# B&R Automation Studio project NAEUL004C00R13L518F00 (part 48)

#### Act_Link.st - Change By Project
```iecst
(** 2019-07-04 **)
ACTION Act_Link:

	//Temporary (Recipe No Save)
	IF p_tyCurrProdRcp.sRcpNm = '' AND p_tyCurrProdRcp.diWidthInUM = 0 THEN
		p_tyCurrProdRcp	:= p_tyInternalReqProdRcp;
	END_IF

	//Info Message
	IF p_eLinkNtParamProjMag = ULMagDual THEN
		bBffrMagRemoved		:= (p_bLinkBffr1MagRemoved = TRUE) AND (p_bLinkBffr2MagRemoved = TRUE);
//		bOpsInitDone		:= ((p_bLinkNtParamProjMagConv1Prep AND p_bLinkOpsMagConvUL1InitDone) OR (NOT p_bLinkNtParamProjMagConv1Prep AND p_bLinkOpsMagUL1InitDone))
//								AND ((p_bLinkNtParamProjMagConv2Prep AND p_bLinkOpsMagConvUL2InitDone) OR (NOT p_bLinkNtParamProjMagConv2Prep AND p_bLinkOpsMagUL2InitDone));
		bOpsInitDone		:= p_bLinkOpsMagConvUL1InitDone AND p_bLinkOpsMagConvUL2InitDone;
	ELSIF p_eLinkNtParamProjMag = ULMagTriple THEN
		bBffrMagRemoved		:= (p_bLinkBffr1MagRemoved = TRUE) AND (p_bLinkBffr2MagRemoved = TRUE) AND (p_bLinkBffr3MagRemoved = TRUE);
//		bOpsInitDone		:= ((p_bLinkNtParamProjMagConv1Prep AND p_bLinkOpsMagConvUL1InitDone) OR (NOT p_bLinkNtParamProjMagConv1Prep AND p_bLinkOpsMagUL1InitDone))
//								AND ((p_bLinkNtParamProjMagConv2Prep AND p_bLinkOpsMagConvUL2InitDone) OR (NOT p_bLinkNtParamProjMagConv2Prep AND p_bLinkOpsMagUL2InitDone))
//								AND ((p_bLinkNtParamProjMagConv3Prep AND p_bLinkOpsMagConvUL3InitDone) OR (NOT p_bLinkNtParamProjMagConv3Prep AND p_bLinkOpsMagUL3InitDone));
		bOpsInitDone		:= p_bLinkOpsMagConvUL1InitDone AND p_bLinkOpsMagConvUL2InitDone AND p_bLinkOpsMagConvUL3InitDone;

	END_IF

	IF bBffrMagRemoved = FALSE THEN
		p_sInfoMsg		:= 'New Recipe Loaded';
		p_sInfoMsg		:= CONCAT(p_sInfoMsg , '$r$n');
		p_sInfoMsg		:= CONCAT(p_sInfoMsg , '$r$n');
		p_sInfoMsg		:= CONCAT(p_sInfoMsg , 'Please Remove All Magazines.');
	ELSE
		p_sInfoMsg		:= '';
	END_IF

	//Accept New Recipe Condition (Before Loaded New Recipe)
	p_bAccNewRcpCond	:=  bBffrMagRemoved = TRUE;

	//Update New Recipe Condition (After Loaded New Recipe)
	p_bUpdtNewRcpCond	:= TRUE;

	//Recipe Different
	p_bInternalReqProdRcpDiff	:= memcmp(ADR(p_tyCurrProdRcp) , ADR(p_tyInternalReqProdRcp) , SIZEOF(p_tyCurrProdRcp)) <> 0;
	p_bUpdtProdRcpDiff			:= memcmp(ADR(p_tyCurrProdRcp) , ADR(tyUpdtProdRcp) , SIZEOF(p_tyCurrProdRcp)) <> 0;

END_ACTION
```

#### Act_InitLocal.st - Do Not Change!!!
```iecst
(** 2020-08-06 **)
ACTION Act_InitLocal:

//Input Reference Link To Local Variable
	p_sMagRcpNm ACCESS ADR(sMagRcpNm);
	p_bUIProdAccData ACCESS ADR(bUIProdAccData);
	p_bUIProdUpdtData ACCESS ADR(bUIProdUpdtData);
	p_bUIMagAccData ACCESS ADR(bUIMagAccData);
	pa_tyProdRcpList ACCESS ADR(a_tyProdRcpList);
	p_tyCurrProdRcp ACCESS ADR(tyCurrProdRcp);
	p_sCurrMagRcpNm ACCESS ADR(sCurrMagRcpNm);
	p_bAccNewRcpCond ACCESS ADR(bAccNewRcpCond);
	p_bUpdtNewRcpCond ACCESS ADR(bUpdtNewRcpCond);
	p_bAutoUpdtData ACCESS ADR(bAutoUpdtData);
	p_sInfoMsg ACCESS ADR(sInfoMsg);
	p_bInternalUse ACCESS ADR(bInternalUse);
	p_tyInternalReqProdRcp ACCESS ADR(tyInternalReqProdRcp);
	p_bNewBrdEnteredCond ACCESS ADR(bNewBrdEnteredCond);
	p_bOldBrdExitedCond ACCESS ADR(bOldBrdExitedCond);
	p_bRlsBrd ACCESS ADR(bRlsBrd);
	p_bInternalReqProdRcpDiff ACCESS ADR(bInternalReqProdRcpDiff);
	p_bUpdtProdRcpDiff ACCESS ADR(bUpdtProdRcpDiff);
	p_bRlsBrdProdRcpDiff ACCESS ADR(bRlsBrdProdRcpDiff);
	p_tyFollower ACCESS ADR(tyFollower);

END_ACTION
```

#### Act_Background.st - Do Not Change!!!
```iecst
(** 2021-05-18 **)
ACTION Act_Background:

	IF p_bInternalUse = TRUE THEN
		tyLeaderToFollowerTag.sReqProdRcpNm		:= p_tyInternalReqProdRcp.sRcpNm;
		IF p_bWidth2Prep THEN
			tyLeaderToFollowerTag.diReqProdRcpWidth	:= p_tyInternalReqProdRcp.diWidthInUM2;
		ELSE
			tyLeaderToFollowerTag.diReqProdRcpWidth	:= p_tyInternalReqProdRcp.diWidthInUM;
		END_IF
		tyLeaderToFollowerTag.sReqMagRcpNm		:= '';
		tyLeaderToFollowerTag.bMnlAccData		:= FALSE;
		tyLeaderToFollowerTag.bBypassMnlAccData	:= FALSE;
		tyLeaderToFollowerTag.bBlkDS			:= FALSE;
		tyLeaderToFollowerTag.bBlkUS			:= FALSE;
		tyLeaderToFollowerTag.bBypassWidthChk	:= TRUE;
		tyLeaderToFollowerTag.bSetTm			:= FALSE;
		tyLeaderToFollowerTag.dtTm				:= 0;
		tyLeaderToFollowerTag.uiTmZone			:= 0;
		tyLeaderToFollowerTag.usiRunTm			:= 0;
		tyLeaderToFollowerTag.bProdNameUSWarn	:= FALSE;
		tyLeaderToFollowerTag.bProdNameDSWarn	:= FALSE;
		tyLeaderToFollowerTag.bProdWidthUSWarn	:= FALSE;
		tyLeaderToFollowerTag.bProdWidthDSWarn	:= FALSE;
		tyLeaderToFollowerTag.bLeaderSeqCtrlInActive	:= FALSE;
	END_IF

	Act_Background_UpdtData;

	//FB
	fbFollower.tyLeaderToFollowerTag	:= tyLeaderToFollowerTag;
	fbFollower.sMcNm					:= p_sMcNm;
	fbFollower.sIPAddr					:= p_sIPAddr;
	fbFollower.bSectionLeader			:= p_bSectionLeader;
	fbFollower.sCurrProdRcpNm			:= p_tyCurrProdRcp.sRcpNm;
	fbFollower.diCurrProdWidthUS		:= p_tyCurrProdRcp.diWidthInUM;
	fbFollower.diCurrProdWidthDS		:= p_tyCurrProdRcp.diWidthInUM2;
	fbFollower.sCurrMagRcpNm			:= p_sCurrMagRcpNm;
	fbFollower.sUpdtLeaderProdRcpNm		:= p_tyToLeaderProdRcp.sRcpNm;
	fbFollower.diUpdtLeaderProdWidthUS	:= p_tyToLeaderProdRcp.diWidthInUM;
	fbFollower.diUpdtLeaderProdWidthDS	:= p_tyToLeaderProdRcp.diWidthInUM2;
	fbFollower.sUpdtLeaderMagRcpNm		:= p_sMagRcpNm;
	fbFollower.bMnlAccDat				:= p_bMnlAccData;
	fbFollower.bAWEn					:= (p_bAWPrep = TRUE) AND (p_bAWDis = FALSE);
	fbFollower.bUSWidthChkEn			:= p_bUSWidthChkPrep AND p_bUSWidthChkEn;
	fbFollower.bUSWidthChkSen			:= p_bUSWidthChkSen;
	fbFollower.bDSWidthChkEn			:= p_bDSWidthChkPrep AND p_bDSWidthChkEn;
	fbFollower.bDSWidthChkSen			:= p_bDSWidthChkSen;
	fbFollower.bProdWidthChk			:= p_bProdWidthChk;
	fbFollower.bProdRcpErr				:= bProdRcpErr;
	fbFollower.bMagRcpErr				:= bMagRcpErr;
	fbFollower.bSetTmErr				:= bSetTmErr;
	fbFollower.eCurrMachineStat			:= eCurrMachineStat;
	fbFollower.bProdChgOverActive		:= (p_eAWStat = AWActGoWidthOff);
	fbFollower.bDBAOnWOAlign			:= p_bDBAOnWOAlign;
	fbFollower(bEn := TRUE);

	tyFollowerToLeaderTag	:= fbFollower.tyFollowerToLeaderTag;
	bProdAccDataReq			:= fbFollower.bProdAccDataReq OR (p_bInternalReqProdRcpDiff = TRUE) ;
	bMagAccDataReq			:= fbFollower.bMagAccDataReq;
	bAutoAccData			:= fbFollower.bAutoAccData;

	IF p_bInternalUse THEN
		bLeaderOnline		:= TRUE;
	ELSE
		bLeaderOnline		:= tyLeaderInfo.bOnline;
	END_IF

	IF bLeaderOnline=FALSE THEN
		bUSAllow				:= TRUE;
		bDSAllow				:= TRUE;
		bLeaderSeqCtrlInActive	:= FALSE;
	ELSE
		bUSAllow				:= fbFollower.bUSAllow AND (p_bInternalReqProdRcpDiff = FALSE);
		bDSAllow				:= fbFollower.bDSAllow;
		bLeaderSeqCtrlInActive	:= tyLeaderToFollowerTag.bLeaderSeqCtrlInActive;
	END_IF

	fbOnlineChk.tyLeaderToFollowerTag	:= tyLeaderToFollowerTag;
	fbOnlineChk(bEn := TRUE);

	Act_Background_AccData;
	Act_Background_ChkRlsBrd;

	//Set Time
	IF EDGEPOS(tyLeaderToFollowerTag.bSetTm) THEN
		bSetTm	:= TRUE;
	END_IF

	IF bSetTm = TRUE THEN
		eTimeAct	:= TimeActSetTime;

		IF (p_eTimeStat = TimeActSetTime) AND (p_eTimeStatus = Done) THEN
			eTimeAct		:= TimeActIdle;
			bSetTm			:= FALSE;
		ELSIF p_eTimeStatus = Error THEN
			eTimeAct		:= TimeActIdle;
			bSetTm			:= FALSE;
		END_IF
	END_IF

	bSetTmErr	:= p_eTimeStatus = Error;

	IF (eStatus = Error) AND bRstErr THEN
		eStatus		:= Idle;
		udiStatus	:= 0;
		bProdRcpErr	:= FALSE;
		bProdRcpErrNotExist	:= FALSE;
		bProdRcpErrWidthMismatch:= FALSE;
		bMagRcpErr	:= FALSE;
	END_IF

END_ACTION
```

#### Act_Background_ChkRlsBrd.st - Do Not Change!!!
```iecst
ACTION Act_Background_ChkRlsBrd:

	IF tyRlsBrdProdRcpNm.sRcpNm = '' THEN
		tyRlsBrdProdRcpNm	:= p_tyCurrProdRcp;

	ELSIF (tyRlsBrdProdRcpNm.sRcpNm <> p_tyCurrProdRcp.sRcpNm) OR (p_bRlsBrdProdRcpDiff = TRUE) THEN

		IF p_bNewBrdEnteredCond = TRUE THEN
			bNewBrdEntered	:= TRUE;
		END_IF

		IF p_bOldBrdExitedCond = TRUE THEN
			bOldBrdExited	:= TRUE;
		END_IF

		IF bNewBrdEntered AND bOldBrdExited THEN
			tylocalFollower.Out.bWaitRlsBrd	:= TRUE;
		END_IF

		IF tylocalFollower.Out.bWaitRlsBrd AND p_bRlsBrd THEN
			tyRlsBrdProdRcpNm	:= p_tyCurrProdRcp;
		END_IF

	ELSE
		bNewBrdEntered	:= FALSE;
		bOldBrdExited	:= FALSE;
		tylocalFollower.Out.bWaitRlsBrd		:= FALSE;

	END_IF

END_ACTION
```

#### Act_Background_AccData.st - Do Not Change!!!
```iecst
ACTION Act_Background_AccData:
	//Product Accept Data Request
	CASE usiProdAccDatStep OF
		0:
			//Check Error & Request Accept Data
			// If Product Name/Width Error, Check In Background To Update Data
			IF ((tylocalFollower.Out.eStatus <> Error) AND (bProdAccDataReq = TRUE)) OR bProdRcpErr THEN
				sReqProdRcpNm		:= tyLeaderToFollowerTag.sReqProdRcpNm;
				diReqProdRcpWidth	:= tyLeaderToFollowerTag.diReqProdRcpWidth;
				usiProdAccDatStep	:= 1;
			END_IF

			IF bLeaderOnline=FALSE THEN
				tyInfoData.udiCode		:= 0;
				tyInfoData.eSeverity	:= AlmSeverityNA;

				bProdRcpErr 			:= FALSE;
				bProdRcpErrNotExist		:= FALSE;
				bProdRcpErrWidthMismatch:= FALSE;
			END_IF

		1:
			IF p_bInternalUse THEN
				usiProdAccDatStep	:= 2;
			ELSE

				//Check In List Of Recipe
				FOR i := 1 TO 2000 DO
					IF sReqProdRcpNm = '' THEN
						EXIT;
					ELSIF sReqProdRcpNm = pa_tyProdRcpList[i].sRcpNm  THEN
						EXIT;
					END_IF
				END_FOR

				IF sReqProdRcpNm = pa_tyProdRcpList[i].sRcpNm AND diReqProdRcpWidth <> pa_tyProdRcpList[i].diWidthInUM THEN
					//Width Mismatch
					bProdRcpErr := TRUE;
					bProdRcpErrWidthMismatch:= TRUE;
					bProdRcpErrNotExist		:= FALSE;
					usiProdAccDatStep	:= 0;
				ELSIF i > 2000 THEN
					//Recipe Not Exist
					bProdRcpErr := TRUE;
					bProdRcpErrNotExist	:= TRUE;
					bProdRcpErrWidthMismatch:= FALSE;
					usiProdAccDatStep	:= 0;
				ELSE
					bProdRcpErr := FALSE;
					bProdRcpErrNotExist	:= FALSE;
					bProdRcpErrWidthMismatch:= FALSE;
					usiProdAccDatStep	:= 2;
				END_IF

				//Info Message
				IF bLeaderOnline=FALSE THEN
					tyInfoData.udiCode		:= 0;
					tyInfoData.eSeverity	:= AlmSeverityNA;

					bProdRcpErr 			:= FALSE;
					bProdRcpErrNotExist		:= FALSE;
					bProdRcpErrWidthMismatch:= FALSE;
				ELSE
					IF p_bInternalUse = FALSE THEN
						IF bLeaderInfo OR bFollowerInfo THEN
//							tyInfoData.sProgNm		:= g_tyNtParamCurr.sFollower1ProgNm;
							tyInfoData.udiCode		:= 10000;
							tyInfoData.eSeverity	:= AlmSeverityInfo;
						ELSE
//							tyInfoData.sProgNm		:= '';
							tyInfoData.udiCode		:= 0;
							tyInfoData.eSeverity	:= AlmSeverityNA;
						END_IF
					ELSE
						IF p_sInfoMsg <> '' THEN
//							tyInfoData.sProgNm		:= g_tyNtParamCurr.sFollower1ProgNm;
							tyInfoData.udiCode		:= 10000;
							tyInfoData.eSeverity	:= AlmSeverityInfo;
						ELSE
//							tyInfoData.sProgNm		:= '';
							tyInfoData.udiCode		:= 0;
							tyInfoData.eSeverity	:= AlmSeverityNA;
							tyInfoData.sAlmMsg		:= '';
						END_IF
					END_IF
				END_IF
			END_IF

		2:
			//Manual Accept Data Check
			IF bProdAccDataReq = TRUE THEN
				IF bAutoAccData = FALSE THEN
				tylocalFollower.Out.bProdAccDataMnl	:= TRUE;

					//Info Message
					IF bLeaderOnline=FALSE THEN
//						tyInfoData.sProgNm		:= '';
						tyInfoData.udiCode		:= 0;
						tyInfoData.eSeverity	:= AlmSeverityNA;
//						tyInfoData.sAlmMsg		:= '';
					ELSE
						IF p_sInfoMsg <> '' THEN
//							tyInfoData.sProgNm		:= g_tyNtParamCurr.sFollower1ProgNm;
							tyInfoData.udiCode		:= 10000;
							tyInfoData.eSeverity	:= AlmSeverityInfo;
//							tyInfoData.sAlmMsg		:= p_sInfoMsg;
						ELSE
//							tyInfoData.sProgNm		:= '';
							tyInfoData.udiCode		:= 0;
							tyInfoData.eSeverity	:= AlmSeverityNA;
//							tyInfoData.sAlmMsg		:= '';
						END_IF
					END_IF

					IF p_bUIProdAccData = TRUE THEN
						tylocalFollower.Out.bProdAccDataMnl		:= FALSE;
						usiProdAccDatStep	:= 3;
					END_IF
				ELSE
					bProdAccDataMnl		:= FALSE;
					tylocalFollower.Out.bProdAccDataMnl		:= FALSE;
					usiProdAccDatStep	:= 3;
				END_IF
			ELSE
				bProdAccDataMnl		:= FALSE;
				usiProdAccDatStep	:= 6;
			END_IF

		3:
			//Accept New Recipe Condition
			IF bProdAccDataReq = TRUE THEN
				IF p_bAccNewRcpCond = TRUE THEN

					usiProdAccDatStep	:= 4;
				ELSE
					//Info Message
					IF bLeaderOnline=FALSE THEN
//						tyInfoData.sProgNm		:= '';
						tyInfoData.udiCode		:= 0;
						tyInfoData.eSeverity	:= AlmSeverityNA;
//						tyInfoData.sAlmMsg		:= '';
					ELSE
						IF p_sInfoMsg <> '' THEN
//							tyInfoData.sProgNm		:= g_tyNtParamCurr.sFollower1ProgNm;
							tyInfoData.udiCode		:= 10000;
							tyInfoData.eSeverity	:= AlmSeverityInfo;
//							tyInfoData.sAlmMsg		:= p_sInfoMsg;
						ELSE
//							tyInfoData.sProgNm		:= '';
							tyInfoData.udiCode		:= 0;
							tyInfoData.eSeverity	:= AlmSeverityNA;
//							tyInfoData.sAlmMsg		:= '';
						END_IF
					END_IF
				END_IF
			ELSE
				usiProdAccDatStep	:= 6;
			END_IF

		4:
			//Accept New Recipe Name
			IF p_bInternalUse = TRUE THEN

				p_tyCurrProdRcp	:= p_tyInternalReqProdRcp;
				usiProdAccDatStep := 6;
			ELSE

				FOR i := 1 TO 2000 DO
					IF sReqProdRcpNm = '' THEN
						EXIT;
					ELSIF sReqProdRcpNm = pa_tyProdRcpList[i].sRcpNm THEN
						p_tyCurrProdRcp	:= pa_tyProdRcpList[i];
						EXIT;
					END_IF
				END_FOR

				IF i > 2000 THEN
					//Recipe Not Exist
					bProdRcpErr := TRUE;
					bProdRcpErrNotExist	:= TRUE;
				END_IF
				usiProdAccDatStep	:= 5;
			END_IF

		5:
			(* Add *)
			p_tyProdRcpCurrRcpWr 	:= p_tyCurrProdRcp;
			p_eLinkUIProdRcpAct 	:= ProdRcpActWriteCurrRcpParam;

			IF p_eProdRcpStat = ProdRcpActWriteCurrRcpParam AND p_eProdRcpStatus = Done THEN
				p_eLinkUIProdRcpAct := ProdRcpActIdle;
				usiProdAccDatStep := 6;
			END_IF

		6:
			//Clear Info Message
			tyInfoData.sProgNm		:= '';
			tyInfoData.udiCode		:= 0;
			tyInfoData.eSeverity	:= AlmSeverityNA;
			tyInfoData.sAlmMsg		:= '';

			usiProdAccDatStep	:= 0;

	END_CASE

END_ACTION
```

#### Act_Main_Disable.st - Do Not Change!!!
```iecst
ACTION Act_Main_Disable:

	tylocalFollower.Out.bUSAllow			:= TRUE;
	tylocalFollower.Out.bDSAllow			:= TRUE;
	tylocalFollower.Out.bProdAccDataMnl		:= FALSE;
	tylocalFollower.Out.bProdUpdtDataMnl	:= FALSE;
	tylocalFollower.Out.bMagAccDataMnl		:= FALSE;
	tylocalFollower.Out.bWaitRlsBrd			:= FALSE;

	usiProdAccDatStep		:= 0;
	usiProdUpdtDatStep		:= 0;
	tyInfoData.udiCode		:= 0;
	tyInfoData.eSeverity	:= AlmSeverityNA;

	usiMagAccDatStep		:= 0;
	tylocalFollower.Out.tyInfoData1.udiCode		:= 0;
	tylocalFollower.Out.tyInfoData1.eSeverity	:= AlmSeverityNA;

	bSetTm		:= FALSE;

	tylocalFollower.Out.eStatus		:= Idle;
	udiStatus	:= 0;
	bProdRcpErr	:= FALSE;
	bMagRcpErr	:= FALSE;
	tylocalFollower.Out.bLdrSeqCtrlInActive	:= FALSE;

	bProdRcpErrNotExist		:= FALSE;
	bProdRcpErrWidthMismatch:= FALSE;

END_ACTION
```

#### Act_Alarm.st - Do Not Change!!!
```iecst
ACTION Act_Alarm:

	IF g_tyRstErrOut.udiRstErr <> udiRstErrOld THEN
		bRstErr			:= TRUE;
		udiRstErrOld	:= g_tyRstErrOut.udiRstErr;
	ELSE
		bRstErr			:= FALSE;
	END_IF

	//Error
	IF EDGEPOS(tylocalFollower.Out.eStatus = Error) THEN

		tylocalFollower.Out.tyAlmData.udiCode		:= udiStatus;
		tylocalFollower.Out.tyAlmData.eSeverity		:= AlmSeverityError;
		tylocalFollower.Out.tyAlmData.udiRunTime	:= tyAlmData.udiRunTime + 1;
		tylocalFollower.Out.tyAlmData.bAlm			:= TRUE;
		tylocalFollower.Out.tyAlmData.udiModuleNum	:= udiModuleNum;
		g_tyAlmProgNm.sLFFollowerProgNm				 := g_tyNtParamCurr.sFollower2ProgNm;

	ELSIF bRstErr AND (tylocalFollower.Out.tyAlmData.udiCode <> 0) THEN

		tylocalFollower.Out.tyAlmData.udiCode	:= 0;
		tylocalFollower.Out.tyAlmData.eSeverity	:= AlmSeverityNA;
		tylocalFollower.Out.tyAlmData.bAlm		:= FALSE;

	END_IF

END_ACTION
```

#### InputRef.var - Do Not Change!!!
```iecst
(*2020-08-06*)
(**)
(*General*)
VAR
	p_udiRstErr : REFERENCE TO UDINT;
	p_bPrep : REFERENCE TO BOOL;
	p_bEn : REFERENCE TO BOOL;
	p_bDis : REFERENCE TO BOOL;
END_VAR
(**)
(*Configuration*)
VAR
	p_eAWStat : REFERENCE TO eAWAction;
	p_sIPAddr : REFERENCE TO STRING[15];
END_VAR
(**)
(*Input*)
VAR
	p_sMcNm : REFERENCE TO STRING[30];
	p_bAWPrep : REFERENCE TO BOOL;
	p_bAWDis : REFERENCE TO BOOL;
	p_bMnlAccData : REFERENCE TO BOOL;
	p_bSectionLeader : REFERENCE TO BOOL;
	p_sMagRcpNm : REFERENCE TO STRING[30];
	p_diWidthLimit : REFERENCE TO DINT;
	p_bWidth2Prep : REFERENCE TO BOOL;
	p_bNtParamAutoRcpPrep : REFERENCE TO BOOL;
	p_bMcParamAutoRcpDis : REFERENCE TO BOOL;
	p_bNtParamAutoRcpF1ArbitraryType : REFERENCE TO BOOL;
	p_bUSWidthChkPrep : REFERENCE TO BOOL;
	p_bUSWidthChkEn : REFERENCE TO BOOL;
	p_bUSWidthChkSen : REFERENCE TO BOOL;
	p_bDSWidthChkPrep : REFERENCE TO BOOL;
	p_bDSWidthChkEn : REFERENCE TO BOOL;
	p_bDSWidthChkSen : REFERENCE TO BOOL;
	p_bProdWidthChk : REFERENCE TO BOOL;
	p_bUIProdAccData : REFERENCE TO BOOL;
	p_bUIProdUpdtData : REFERENCE TO BOOL;
	p_bUIMagAccData : REFERENCE TO BOOL;
	pa_tyProdRcpList : REFERENCE TO ARRAY[1..c_udiProdRcpMax] OF tyProdRcpParam;
	p_tyCurrProdRcp : REFERENCE TO tyProdRcpParam;
	p_sCurrMagRcpNm : REFERENCE TO STRING[30];
	p_eTimeStat : REFERENCE TO eTimeAction;
	p_eTimeStatus : REFERENCE TO eFBStatus;
	p_bAccNewRcpCond : REFERENCE TO BOOL;
	p_bUpdtNewRcpCond : REFERENCE TO BOOL;
	p_bAutoUpdtData : REFERENCE TO BOOL;
	p_sInfoMsg : REFERENCE TO STRING[200];
	p_bInternalUse : REFERENCE TO BOOL;
	p_tyInternalReqProdRcp : REFERENCE TO tyProdRcpParam;
	p_bNewBrdEnteredCond : REFERENCE TO BOOL;
	p_bOldBrdExitedCond : REFERENCE TO BOOL;
	p_bRlsBrd : REFERENCE TO BOOL;
	p_tyToLeaderProdRcp : REFERENCE TO tyProdRcpParam;
	p_bInternalReqProdRcpDiff : REFERENCE TO BOOL;
	p_bUpdtProdRcpDiff : REFERENCE TO BOOL;
	p_bRlsBrdProdRcpDiff : REFERENCE TO BOOL;
	p_sProgNm : REFERENCE TO STRING[15];
	p_bNtSettingsLoadDone : REFERENCE TO BOOL;
	p_tOnlineChkDlyTm : REFERENCE TO TIME;
	p_bManual : REFERENCE TO BOOL;
	p_bErr : REFERENCE TO BOOL;
	p_bWarning : REFERENCE TO BOOL;
	p_bOps : REFERENCE TO BOOL;
	p_bStandby : REFERENCE TO BOOL;
	p_bDBAOnWOAlign : REFERENCE TO BOOL;
END_VAR
```

#### Local.var - Do Not Change!!!
```iecst
VAR
	tylocalFollower : tyLFFollower1;
END_VAR
(**)
VAR
	udiStatus : UDINT := 0;
END_VAR
(**)
(*Local Alarm*)
VAR
	tyAlmData : tyAlmDat;
	tyInfoData : tyAlmDat;
	tyInfoData1 : tyAlmDat;
END_VAR
(**)
VAR
	sMagRcpNm : STRING[30];
	bUIProdAccData : BOOL;
	bUIProdUpdtData : BOOL;
	bUIMagAccData : BOOL;
	a_tyProdRcpList : ARRAY[1..c_udiProdRcpMax] OF tyProdRcpParam;
	tyDispProdRcp : tyProdRcpParam;
	tyCurrProdRcp : tyProdRcpParam;
	sCurrMagRcpNm : STRING[30];
	bAccNewRcpCond : BOOL;
	bUpdtNewRcpCond : BOOL;
	bAutoUpdtData : BOOL;
	sInfoMsg : STRING[200];
	bInternalUse : BOOL;
	tyInternalReqProdRcp : tyProdRcpParam;
	bNewBrdEnteredCond : BOOL;
	bOldBrdExitedCond : BOOL;
	bRlsBrd : BOOL;
	tyToLeaderProdRcp : tyProdRcpParam;
	bInternalReqProdRcpDiff : BOOL;
	bUpdtProdRcpDiff : BOOL;
	bRlsBrdProdRcpDiff : BOOL;
	sWidthInUMTemp : STRING[80];
END_VAR
(**)
(*Local*)
VAR
	bRstErr : BOOL;
	udiRstErrOld : UDINT;
	bInitDone : BOOL;
	bInitialDone : BOOL;
	bAutoAccData : BOOL;
	bProdRcpErr : BOOL;
	bMagRcpErr : BOOL;
	bSetTmErr : BOOL;
	bProdAccDataReq : BOOL;
	sReqProdRcpNm : STRING[254];
	diReqProdRcpWidth : DINT;
	bMagAccDataReq : BOOL;
	sReqMagRcpNm : STRING[30];
	usiProdAccDatStep : USINT;
	usiMagAccDatStep : USINT;
	usiProdUpdtDatStep : USINT;
	tyRlsBrdProdRcpNm : tyProdRcpParam;
	bNewBrdEntered : BOOL;
	bOldBrdExited : BOOL;
	i : INT;
	bSetTm : BOOL;
	fbOnlineChk : fbLFFollowerOnlineChk;
	fbFollower : fbLFFollower;
	tyLeaderToFollowerTag : tyLFLeaderToFollowerTag;
	tyFollowerToLeaderTag : tyLFFollowerToLeaderTag;
	eCurrMachineStat : eMachineStat;
	bLeaderOnline : BOOL;
	bLeaderInfo : BOOL;
	bFollowerInfo : BOOL;
	bProdRcpErrNotExist : BOOL;
	bProdRcpErrWidthMismatch : BOOL;
	tyFollower : {REDUND_UNREPLICABLE} tyLFFollowerOut1;
	bBffrMagRemoved : BOOL;
	bOpsInitDone : BOOL;
END_VAR
(**)
VAR
	p_sMagRcpNm : REFERENCE TO STRING[30];
	p_bUIProdAccData : REFERENCE TO BOOL;
	p_bUIProdUpdtData : REFERENCE TO BOOL;
	p_bUIMagAccData : REFERENCE TO BOOL;
	pa_tyProdRcpList : REFERENCE TO ARRAY[1..c_udiProdRcpMax] OF tyProdRcpParam;
	p_tyCurrProdRcp : REFERENCE TO tyProdRcpParam;
	p_tyDispProdRcp : REFERENCE TO tyProdRcpParam;
	p_sCurrMagRcpNm : REFERENCE TO STRING[30];
	p_bAccNewRcpCond : REFERENCE TO BOOL;
	p_bUpdtNewRcpCond : REFERENCE TO BOOL;
	p_bAutoUpdtData : REFERENCE TO BOOL;
	p_sInfoMsg : REFERENCE TO STRING[200];
	p_bInternalUse : REFERENCE TO BOOL;
	p_tyInternalReqProdRcp : REFERENCE TO tyProdRcpParam;
	p_bNewBrdEnteredCond : REFERENCE TO BOOL;
	p_bOldBrdExitedCond : REFERENCE TO BOOL;
	p_bRlsBrd : REFERENCE TO BOOL;
	p_bInternalReqProdRcpDiff : REFERENCE TO BOOL;
	p_bUpdtProdRcpDiff : REFERENCE TO BOOL;
	p_bRlsBrdProdRcpDiff : REFERENCE TO BOOL;
	p_tyFollower : REFERENCE TO tyLFFollowerOut1;
	udiModuleNum : UDINT := 3901;
END_VAR
```

#### Act_InputConfig.st - not listed in the package file held
```iecst
(** 2019-06-12 **)
ACTION Act_InputConfig:

	(* Always Change If Project Change *)

	//Pass Data To Internal Use

	p_tyCurrProdRcp ACCESS p_ProdRcpCurrRcp2;
	p_tyInternalReqProdRcp ACCESS p_ProdRcpCurrRcp1;	//Follower 2 Assign With Follower 1 Recipe

	tylocalFollower.In.bDis	:= (g_tyStartUp.bRun = TRUE);
	tylocalFollower.In.bPrep := NOT(g_tyNtParamCurr.bAutoRcpPrep) OR g_tyMcParamCurr.bAutoRcpDisable;

	//Temporary (Recipe No Save)
	IF p_tyCurrProdRcp.sRcpNm = '' AND p_tyCurrProdRcp.diWidthInUM = 0 THEN
		p_tyCurrProdRcp	:= p_tyInternalReqProdRcp;
	END_IF

	//Info Message
	IF g_tyNtParamCurr.eProjMag = ULMagDual THEN
		bBffrMagRemoved		:= (g_tyBuffer1.bMagRemoved = TRUE) AND (g_tyBuffer2.bMagRemoved = TRUE);
		bOpsInitDone		:= g_tyOpsMagConvUL1.bInitDone AND g_tyOpsMagConvUL2.bInitDone;
	ELSIF g_tyNtParamCurr.eProjMag = ULMagTriple THEN
		bBffrMagRemoved		:= (g_tyBuffer1.bMagRemoved = TRUE) AND (g_tyBuffer2.bMagRemoved = TRUE) AND (g_tyBuffer3.bMagRemoved = TRUE);
		bOpsInitDone		:= g_tyOpsMagConvUL1.bInitDone AND g_tyOpsMagConvUL2.bInitDone AND g_tyOpsMagConvUL3.bInitDone;
	END_IF

	IF bBffrMagRemoved = FALSE THEN
		p_sInfoMsg		:= 'New Recipe Loaded';
		p_sInfoMsg		:= CONCAT(p_sInfoMsg , '$r$n');
		p_sInfoMsg		:= CONCAT(p_sInfoMsg , '$r$n');
		p_sInfoMsg		:= CONCAT(p_sInfoMsg , 'Please Remove All Magazines.');
	ELSE
		p_sInfoMsg		:= '';
	END_IF

	//Accept New Recipe Condition (Before Loaded New Recipe)
	p_bAccNewRcpCond	:=  bBffrMagRemoved = TRUE;

	//Update New Recipe Condition (After Loaded New Recipe)
	p_bUpdtNewRcpCond	:= TRUE;

	//Recipe Different
	p_bInternalReqProdRcpDiff	:= memcmp(ADR(p_tyCurrProdRcp) , ADR(p_tyInternalReqProdRcp) , SIZEOF(p_tyCurrProdRcp)) <> 0;
	p_bUpdtProdRcpDiff			:= memcmp(ADR(p_tyCurrProdRcp) , ADR(tyUpdtProdRcp) , SIZEOF(p_tyCurrProdRcp)) <> 0;

END_ACTION
```

### Follower2.var - not listed in the package file held
```iecst
(*2019-06-27*)
(**)
(*Action & State & Status*)
VAR
	p_Follower2Status : UDINT;
END_VAR
(**)
(*Alarm*)
VAR
	p_Follower2AlmData : UDINT;
	p_Follower2InfoData : UDINT;
	p_Follower2InfoData1 : UDINT;
END_VAR
(**)
(*Output*)
VAR
	p_Follower2USAllow : UDINT;
	p_Follower2DSAllow : UDINT;
	p_Follower2ProdAccDataMnl : UDINT;
	p_Follower2ProdUpdtDataMnl : UDINT;
	p_Follower2MagAccDataMnl : UDINT;
	p_Follower2TimeAct : UDINT;
	p_Follower2SetDT : UDINT;
	p_Follower2WaitRlsBrd : UDINT;
	p_Follower2UpdtProdRcp : UDINT;
	p_Follower2ProdRcpDiff : UDINT;
END_VAR
```

### Machine.typ - Do Not Change!!!
```iecst
TYPE
	tyMachine : 	STRUCT
		In : tyMachineIn1;
		Out : tyMachineOut1;
	END_STRUCT;
	tyMachineIn1 : 	STRUCT
		udiRstErr : UDINT := 0;
		sProgNm : STRING[15];
		diProdRcpCurrRcpWidth : REFERENCE TO DINT;
		diMagRcpCurrRcpMaxWidth : REFERENCE TO DINT;
	END_STRUCT;
	tyMachineOut1 : 	STRUCT
		tyAlmData : tyAlmDat;
		tyAlmData1 : tyAlmDat;
	END_STRUCT;
END_TYPE
```

### Machine.var - Change By Project
```iecst
(*2018-12-07*)
(**)
(*Action & State & Status*)
VAR
	g_tyMachine : tyMachineOut1;
END_VAR
```

### Program Logical/Machine/Machine (IEC, version 1.00.0) - 1.00.0 - 

#### Act_InputConfig.st - Change By Project
```iecst
(** 2019-04-09 **)
ACTION Act_InputConfig:

	(* Always Change If Project Change *)

	//Pass Data To Link

	//Pass Data To Internal Use

	tylocalMachine.In.udiRstErr := g_tyRstErrOut.udiRstErr;
	tylocalMachine.In.diProdRcpCurrRcpWidth ACCESS p_ProdRcpCurrRcp0Width;
	tylocalMachine.In.diMagRcpCurrRcpMaxWidth ACCESS p_MagRcpCurrRcpMagMaxBrdWidth;
	tylocalMachine.In.sProgNm := g_tyNtParamCurr.sMcParamProgNm;

	(* Always Change If Project Change *)

END_ACTION
```

#### Act_OutputConfig.st - Change By Project
```iecst
(** 2019-03-22 **)
ACTION Act_OutputConfig:

	g_tyMachine := tylocalMachine.Out;

END_ACTION
```

#### Cyclic.st - Change By Project
```iecst
(** 2019-03-22 **)
PROGRAM _CYCLIC

	IF bInitialDone = FALSE THEN
		//Special Case --> only after reading Current Recipe --> Excusively for Machine with Magazine Maximum Board Width Setting
		IF g_tyStartUp.bNtSettingsLoadDone = TRUE AND Step = g_tyStartUp.eStartupStep1 =StartupStepUsrMgmt  THEN
			bInitialDone	:= TRUE;
			Act_Initial;
		END_IF

	ELSE

		Act_Background;
		Act_Alarm;
		Act_AlarmInfo1;

	END_IF

END_PROGRAM
```

#### Act_Background.st - Change By Project
```iecst
(** 2019-01-23 **)
ACTION Act_Background:

	IF (tylocalMachine.In.diProdRcpCurrRcpWidth > tylocalMachine.In.diMagRcpCurrRcpMaxWidth) AND (tylocalMachine.Out.eStatus <> Error) THEN
		tylocalMachine.Out.eStatus		:= Error;
		udiStatus   := 10000;
	END_IF

	//Reset Error
	IF (tylocalMachine.Out.eStatus = Error) AND bRstErr THEN
		tylocalMachine.Out.eStatus		:= Idle;
		udiStatus	:= 0;
	END_IF

END_ACTION
```

#### Act_Alarm.st - Change By Project
```iecst
(** 2019-03-25 **)
ACTION Act_Alarm:

	IF tylocalMachine.In.udiRstErr <> udiRstErrOld THEN
		bRstErr			:= TRUE;
		udiRstErrOld	:= tylocalMachine.In.udiRstErr;
	ELSE
		bRstErr			:= FALSE;
	END_IF
	//Error
	IF EDGEPOS(tylocalMachine.Out.eStatus = Error) THEN

		tylocalMachine.Out.tyAlmData.udiCode		:= udiStatus;
		tylocalMachine.Out.tyAlmData.eSeverity		:= AlmSeverityError;
		tylocalMachine.Out.tyAlmData.udiRunTime	:= tylocalMachine.Out.tyAlmData.udiRunTime + 1;
		tylocalMachine.Out.tyAlmData.bAlm			:= TRUE;
		tylocalMachine.Out.tyAlmData.udiModuleNum  := udiModuleNum;
		g_tyAlmProgNm.sMachineProgNm		    := tylocalAGV.In.sProgNm;

		tylocalMachine.Out.sStatTxt	:= tylocalMachine.Out.tyAlmData.sAlmMsg;

	ELSIF bRstErr AND (tyAlmData.udiCode <> 0) THEN

		tylocalMachine.Out.tyAlmData.udiCode	:= 0;
		tylocalMachine.Out.tyAlmData.eSeverity	:= AlmSeverityNA;
		tylocalMachine.Out.tyAlmData.bAlm			:= FALSE;
		tylocalMachine.Out.sStatTxt	:= a_sStatText[tylocalMachine.Out.eStat];

	END_IF

END_ACTION
```

#### Act_AlarmInfo1.st - Do Not Change!!!
```iecst
(** 2019-03-25 **)
ACTION Act_AlarmInfo1:

	//Info

	tylocalMachine.Out.tyAlmData1.udiCode		:= udiStatus1;
	tylocalMachine.Out.tyAlmData1.eSeverity		:= AlmSeverityInfo;
	tylocalMachine.Out.tyAlmData1.udiRunTime	:= tylocalMachine.Out.tyAlmData1.udiRunTime + 1;
	g_tyAlmProgNm.sMachineProgNm		  		  := tylocalMachine.In.sProgNm;
//	//Get Info Message
//	IF tylocalMachine.Out.tyAlmData1.udiCode < 10000 OR tylocalMachine.Out.tyAlmData1.udiCode > 10099 THEN
//		tylocalMachine.Out.tyAlmData1.sAlmMsg	:= 'Unknown';
//		tylocalMachine.Out.tyAlmData1.sRcyMsg	:= 'Unknown';
//	ELSE
//		tylocalMachine.Out.tyAlmData1.sAlmMsg	:= a_tyAlmText[tylocalMachine.Out.tyAlmData1.udiCode].sAlmText;
//		tylocalMachine.Out.tyAlmData1.sRcyMsg	:= a_tyAlmText[tylocalMachine.Out.tyAlmData1.udiCode].sRcyText;
//	END_IF

END_ACTION
```

#### Local.var - Change By Project
```iecst
(*2019-03-25*)
VAR
	tylocalMachine : tyMachine;
END_VAR
(**)
(*Local Action, State & Status*)
VAR
	eStatus : eFBStatus := Idle;
	udiStatus : UDINT := 0;
	udiStatus1 : UDINT := 0;
END_VAR
(**)
(*Local Alarm*)
VAR
	tyAlmData : tyAlmDat;
	tyAlmData1 : tyAlmDat;
	a_tyAlmText : ARRAY[10000..10099] OF tyAlmTxt := [(sAlmText:='Selected Product Width Exceeds Selected Magazine Maximum Board Width',sRcyText:='Please Reselect  Product or Magazine '),99((0))];
END_VAR
(**)
(*Local Output*)
(**)
(*Local Input*)
VAR
	udiRstErr : UDINT := 0;
END_VAR
(**)
VAR
	bOpsRun : BOOL;
	diProdRcpCurrRcpWidth : DINT;
	diMagRcpCurrRcpMaxWidth : DINT;
END_VAR
(**)
VAR
	sProgNm : STRING[15] := 'Machine';
	bNtSettingsLoadDone : BOOL := TRUE;
END_VAR
(**)
(*Local*)
VAR
	bRstErr : BOOL;
	udiRstErrOld : UDINT;
	bInitDone : BOOL;
	bInitialDone : BOOL;
	udiModuleNum : UDINT := 5951;
END_VAR
```

#### InputRef.var - not listed in the package file held
```iecst
(*2019-03-22*)
(**)
(*General*)
VAR
	p_udiRstErr : REFERENCE TO UDINT;
END_VAR
(**)
(*Configuration*)
VAR
	p_bOpsRun : REFERENCE TO BOOL;
	p_bDIPressureSW : REFERENCE TO BOOL;
	p_diProdRcpCurrRcpWidth : REFERENCE TO DINT;
	p_diMagRcpCurrRcpMaxWidth : REFERENCE TO DINT;
	p_eStartupStep : REFERENCE TO eStartupStep;
END_VAR
(**)
VAR
	p_sProgNm : REFERENCE TO STRING[15];
	p_bNtSettingsLoadDone : REFERENCE TO BOOL;
END_VAR
```

#### Act_InitGlobal.st - not listed in the package file held
```iecst
(** 2019-04-09 **)
ACTION Act_InitGlobal:

	(* Always Change If Project Change *)

	//Pass Data To Link

	//Pass Data To Internal Use
	p_udiRstErr ACCESS p_RstErrReset;

	p_bOpsRun ACCESS p_OpsRun;
	p_diProdRcpCurrRcpWidth ACCESS p_ProdRcpCurrRcp0Width;
	p_diMagRcpCurrRcpMaxWidth ACCESS p_MagRcpCurrRcpMagMaxBrdWidth;

	p_eStartupStep ACCESS p_StartupStep;

	p_sProgNm ACCESS p_NtParamMcProgNm;
	p_bNtSettingsLoadDone ACCESS p_StartupNtSettingsLoadDone;

	(* Always Change If Project Change *)

END_ACTION
```

#### Act_InitLocal.st - not listed in the package file held
```iecst
(** 2019-03-25 **)
ACTION Act_InitLocal:

	//Input Reference Link To Local Variable
	p_udiRstErr ACCESS ADR(udiRstErr);

	p_bOpsRun ACCESS ADR(bOpsRun);
	p_diProdRcpCurrRcpWidth ACCESS ADR(diProdRcpCurrRcpWidth);
	p_diMagRcpCurrRcpMaxWidth ACCESS ADR(diMagRcpCurrRcpMaxWidth);

	p_sProgNm ACCESS ADR(sProgNm);
	p_bNtSettingsLoadDone ACCESS ADR(bNtSettingsLoadDone);

END_ACTION
```

#### Init.st - not listed in the package file held
```iecst
(** 2019-03-22 **)
PROGRAM _INIT

	(* Always Change If Project Change *)

	//Pass Address To Global Address For External Use
	//Action, State & Status

	//Alarm
	p_McAlmData		:= ADR(tyAlmData);
	p_McInfoData1	:= ADR(tyAlmData1);

	//Output

	(* Always Change If Project Change *)

END_PROGRAM
```

### AGV.typ - Do Not Change!!!
```iecst
(*2018-12-13*)
(**)
(*Action*)

TYPE
	eAGVMagAction :
		(
		AGVMagActIdle,
		AGVMagActEnter,
		AGVMagActExit
		);
	tyTagDTMagToAGV : 	STRUCT
		bEStopErr : BOOL;
		bCI1MagazineFull : BOOL;
		bCI1Rdy : BOOL;
		bCI1Auto : BOOL;
		bCI1Occupied : BOOL;
		bCI1Running : BOOL;
		bCI1IncorrectMagazineModel : BOOL;
		bCI2MagazineFull : BOOL;
		bCI2Rdy : BOOL;
		bCI2Auto : BOOL;
		bCI2Occupied : BOOL;
		bCI2Running : BOOL;
		bCI2IncorrectMagazineModel : BOOL;
		bCI3MagazineFull : BOOL;
		bCI3Rdy : BOOL;
		bCI3Auto : BOOL;
		bCI3Occupied : BOOL;
		bCI3Running : BOOL;
		bCI3IncorrectMagazineModel : BOOL;
		bCI4MagazineFull : BOOL;
		bCI4Rdy : BOOL;
		bCI4Auto : BOOL;
		bCI4Occupied : BOOL;
		bCI4Running : BOOL;
		bCI4IncorrectMagazineModel : BOOL;
	END_STRUCT;
	tyTagAGVToDTMag : 	STRUCT
		bVEHInPos1 : BOOL;
		bVEHInPos2 : BOOL;
		bVEHInPos3 : BOOL;
		bVEHAuto : BOOL;
		bVEH1Occupied : BOOL;
		bVEH2Occupied : BOOL;
		bVEH3Occupied : BOOL;
		bVEHRunning : BOOL;
	END_STRUCT;
	tyStatToMES : 	STRUCT
		sMachineName : STRING[30];
		bActive : BOOL;
		bAuto_Run : BOOL;
		bError : BOOL;
		bWarning : BOOL;
		nNumberOfPlatforms : USINT;
		tyTagStatOfPlatforms : ARRAY[1..4]OF tyStatPlatform;
	END_STRUCT;
	tyStatFromMES : 	STRUCT
		sMESName : STRING[30];
		bActive : BOOL;
		tyTagStatOfPlatforms : ARRAY[1..4]OF tyStatPlatformFromMES;
	END_STRUCT;
	tyStatPlatform : 	STRUCT
		bMagLoaded : BOOL;
		bError : BOOL;
		bSizeLarge : BOOL;
		bReady : BOOL;
		bAvailable : BOOL;
		bReqAIVToBring : BOOL;
		bReqAIVToGet : BOOL;
		bReadRFID : BOOL;
		bWriteRFID : BOOL;
	END_STRUCT;
	tyStatPlatformFromMES : 	STRUCT
		iAcceptCondition : INT;
		bError : BOOL;
		bSizeLarge : BOOL;
		bReady : BOOL;
		bAvailable : BOOL;
		bRFIDWriteComplete : BOOL;
		bTrigMagFull : BOOL;
	END_STRUCT;
END_TYPE

(*AGV Batch Counting With No Vertical Communication*)

TYPE
	tyStatFromLoader : 	STRUCT
		tyTagStatOfPlatForms : ARRAY[1..4]OF tyStatPlatformFromLoader;
	END_STRUCT;
	tyStatPlatformFromLoader : 	STRUCT
		usiMagBrdUnloadCnt : USINT;
		bFinishedLoading : BOOL;
	END_STRUCT;
END_TYPE

(*AGV Comm in/out*)

TYPE
	tyAGVCom : 	STRUCT
		In : tyAGVComIn1;
		Out : tyAGVComOut1;
	END_STRUCT;
	tyAGVComIn1 : 	STRUCT
		bManual : BOOL;
		tyDTMagToAGV1 : tyTagDTMagToAGV;
		tyDTMagToAGV2 : tyTagDTMagToAGV;
		tyDTMagToAGV3 : tyTagDTMagToAGV;
		bOpsRun : BOOL;
		bLinkOpsSimu : BOOL;
		bIncorrectMagazine1 : BOOL;
		bIncorrectMagazine2 : BOOL;
		bIncorrectMagazine3 : BOOL;
		bRequestToBring1 : BOOL;
		bRequestToBring2 : BOOL;
		bRequestToBring3 : BOOL;
		bRequestToBring4 : BOOL;
		bRequestToGet1 : BOOL;
		bRequestToGet2 : BOOL;
		bRequestToGet3 : BOOL;
		bRequestToGet4 : BOOL;
		bUISOTMagError1 : BOOL;
		bUISOTMagError2 : BOOL;
		bUISOTMagError3 : BOOL;
		bUISOTMagReady1 : BOOL;
		bUISOTMagReady2 : BOOL;
		bUISOTMagReady3 : BOOL;
		bUISOTMagAvailable1 : BOOL;
		bUISOTMagAvailable2 : BOOL;
		bUISOTMagAvailable3 : BOOL;
		bUISOTMagSizeLarge1 : BOOL;
		bUISOTMagSizeLarge2 : BOOL;
		bUISOTMagSizeLarge3 : BOOL;
		bUIRequestToBring1 : BOOL;
		bUIRequestToBring2 : BOOL;
		bUIRequestToBring3 : BOOL;
		bUIRequestToGet1 : BOOL;
		bUIRequestToGet2 : BOOL;
		bUIRequestToGet3 : BOOL;
		bDIFleetManagerActive : BOOL;
		eAGVComProtocol : eMcAGVCommProtocol;
		bSOTMagError1 : BOOL;
		bSOTMagSizeLarge1 : BOOL;
		bSOTMagReady1 : BOOL;
		bSOTMagAvailable1 : BOOL;
		bSOTMagError2 : BOOL;
		bSOTMagSizeLarge2 : BOOL;
		bSOTMagReady2 : BOOL;
		bSOTMagAvailable2 : BOOL;
		bSOTMagError3 : BOOL;
		bSOTMagSizeLarge3 : BOOL;
		bSOTMagReady3 : BOOL;
		bSOTMagAvailable3 : BOOL;
		bAGVSimulationOn : BOOL;
		bDisableFMWarning : BOOL;
		bAGVRdyEnter2 : BOOL;
		bAGVRdyExit2 : BOOL;
		bAGVRdyEnter3 : BOOL;
		bAGVRdyExit3 : BOOL;
		bAGVRdyEnter1 : BOOL;
		bAGVRdyExit1 : BOOL;
		sJobNo : STRING[30];
		sProgNm : STRING[15];
		udiRstErr : UDINT;
		bPrep : BOOL;
		bEn : BOOL;
		bDis : BOOL;
		eCustomerReq : eCustomer;
		bOpsMagConvUL1ReadRFID : BOOL;
		bOpsMagConvUL1WriteRFID : BOOL;
		bOpsMagConvUL2ReadRFID : BOOL;
		bOpsMagConvUL2WriteRFID : BOOL;
		bOpsMagConvUL3ReadRFID : BOOL;
		bOpsMagConvUL3WriteRFID : BOOL;
		tyUIAGVToDTMagSimulateData : tyTagAGVToDTMag;
	END_STRUCT;
	tyAGVComOut1 : 	STRUCT
		eStat : eAGVMagAction;
		eStatus : eFBStatus;
		sStatTxt : STRING[200];
		tyAlmData : tyAlmDat;
		tyAlmData1 : tyAlmDat;
		tyAGVToDTMag : tyTagAGVToDTMag;
		bInternalAGVOnline : BOOL;
		bMachineOnline : BOOL;
		tyDTMagToAGV : tyTagDTMagToAGV;
		bInternalAGVSimulateOn : BOOL;
		tyTagToMes : tyStatToMES;
		tyTagFromMes : tyStatFromMES;
		bFleetManagerActive : BOOL;
	END_STRUCT;
END_TYPE

(*AGV Plat Comm in/out*)

TYPE
	tyAGV1 : 	STRUCT
		In : tyAGVIn1;
		Out : tyAGVOut1;
	END_STRUCT;
	tyAGVIn1 : 	STRUCT
		udiRstErr : UDINT := 0;
		bPrep : BOOL := TRUE;
		bEn : BOOL := TRUE;
		bDis : BOOL := FALSE;
		sProgNm : STRING[15] := 'AIVMag';
		bNtSettingsLoadDone : BOOL := TRUE;
		diTxInTimeOut : DINT;
		diTxOutTimeOut : DINT;
		eDirection : eConvDir;
		bBufferMagPresent : BOOL;
		bMagConvLftSen : BOOL;
		bMagConvRgtSen : BOOL;
		bMagConvMtrIn : BOOL;
		bMagConvMtrOut : BOOL;
		bAGVInPosSen1 : BOOL;
		bAGVInPosSen2 : BOOL;
		bNtParamAGVInPosSenPrep : BOOL;
		bSOTRcvOk : BOOL;
		bSOTErr : BOOL;
		bSOTRdy : BOOL;
		bSOTAvailable : BOOL;
		tyAGVToDTMag : tyTagAGVToDTMag;
		tyDTMagToAGV : tyTagDTMagToAGV;
		bLinkAGVOnline : BOOL;
	END_STRUCT;
	tyAGVOut1 : 	STRUCT
		eStat : eAGVMagAction;
		eStatus : eFBStatus;
		sStatTxt : STRING[200];
		tyAlmData : tyAlmDat;
		bRdyEnt : BOOL;
		bRdyExit : BOOL;
		bMcRunRdy : BOOL;
		tyDTMagToAGV : tyTagDTMagToAGV;
	END_STRUCT;
END_TYPE
```

### AGV.var - Change By Project
```iecst
(*AGV Comm*)
VAR
	g_tyAGV : tyAGVComOut1;
END_VAR
(*AGV pos*)
VAR
	g_tyAGV1 : tyAGVOut1;
	g_tyAGV2 : tyAGVOut1;
	g_tyAGV3 : tyAGVOut1;
END_VAR
```

### Program Logical/AGVCom/AGV (IEC, version 1.00.0) - 1.00.0 - NtSMEMA v5.00.0

#### Act_InputConfig.st - Change By Project
```iecst
(** 2018-12-08 **)
ACTION Act_InputConfig:

	(* Always Change If Project Change *)

	//Pass Data To Linkg_tyMcParamCurr
	tylocalAGV.In.bLinkSafetyRlySig := g_tyDInput.bSafetyRlySig;
	tylocalAGV.In.bLinkCoverSWSig := g_tyDInput.bCoverSWSig;
	tylocalAGV.In.bLinkAlarmWarning := g_tyAlm.bWarning;
	tylocalAGV.In.bLinkAlarmInfo := g_tyAlm.bInfo;
	tylocalAGV.In.bLinkError := g_tyAlm.bErr;
	tylocalAGV.In.eLinkULMag := g_tyNtParamCurr.eProjMag;
	tylocalAGV.In.eLinkAGVComProtocol := g_tyMcParamCurr.eAGVComProtocol;

	//Pass Data To Internal Use

	tylocalAGV.In.bManual := g_tyUIOut.bManualMod;
	tylocalAGV.In.bPrep := g_tyNtParamCurr.bProjAGVPrep;
	tylocalAGV.In.tyDTMagToAGV1 := g_tyAGVMag1.b.tyDTMagToAGV;
	tylocalAGV.In.tyDTMagToAGV2 := g_tyAGVMag2.b.tyDTMagToAGV;
	tylocalAGV.In.tyDTMagToAGV3 := g_tyAGVMag3.b.tyDTMagToAGV;
	tylocalAGV.In.udiRstErr	:= g_tyRstErr.udiReset;
	tylocalAGV.In.sProgNm := g_tyNtParamCurr.sAGVProgNm;
	tylocalAGV.In.bIncorrectMagazine1 := g_tyOpsMagConvUL1.bIncorrectMagModel;
	tylocalAGV.In.bIncorrectMagazine2 := g_tyOpsMagConvUL2.bIncorrectMagModel;
	tylocalAGV.In.bIncorrectMagazine3 := g_tyOpsMagConvUL3.bIncorrectMagModel;

	tylocalAGV.In.tyUIAGVToDTMagSimulateData := g_tyUIOut.tyAGVSimulateSig;
	tylocalAGV.In.bUIAGVOnline := g_tyUIOut.bAGVSimulateOnline;
	tylocalAGV.In.bUIAGVSimulationOn := g_tyUIOut.bAGVSimulationOn;

	tylocalAGV.In.sJobNo := g_tyNtParamCurr.sJobNo;

	tylocalAGV.In.bAGVRdyEnter1 := g_tyAGVMag1.bRdyEnter;
	tylocalAGV.In.bAGVRdyExit1 := g_tyAGVMag1.bRdyExit;
	tylocalAGV.In.bAGVRdyEnter2 := g_tyAGVMag2.bRdyEnter;
	tylocalAGV.In.bAGVRdyExit2 := g_tyAGVMag2.bRdyExit;
	tylocalAGV.In.bAGVRdyEnter3 := g_tyAGVMag3.bRdyEnter;
	tylocalAGV.In.bAGVRdyExit3 := g_tyAGVMag3.bRdyExit;

	tylocalAGV.In.bDIFleetManagerActive := g_tyDInput.bFleetManagerReady;

	tylocalAGV.In.bUISOTMagError1	:= g_tyUIOut.bSOTMagErr1;
	tylocalAGV.In.bUISOTMagError2	:= g_tyUIOut.bSOTMagErr2;
	tylocalAGV.In.bUISOTMagError3	:= g_tyUIOut.bSOTMagErr3;
	//		tylocalAGV.In.bSOTMagError4	:= g_tyUIOut.bSOTMagErr4;
	tylocalAGV.In.bUISOTMagReady1	:= g_tyUIOut.bSOTMagRdy1;
	tylocalAGV.In.bUISOTMagReady2	:= g_tyUIOut.bSOTMagRdy2;
	tylocalAGV.In.bUISOTMagReady3	:= g_tyUIOut.bSOTMagRdy3;
	//		tylocalAGV.In.bSOTMagReady4	:= g_tyUIOut.bSOTMagRdy4;
	tylocalAGV.In.bUISOTMagAvailable1	:= g_tyUIOut.bSOTMagAvail1;
	tylocalAGV.In.bUISOTMagAvailable2	:= g_tyUIOut.bSOTMagAvail2;
	tylocalAGV.In.bUISOTMagAvailable3	:= g_tyUIOut.bSOTMagAvail3;
	//		tylocalAGV.In.bSOTMagAvailable4	:= g_tyUIOut.bSOTMagAvail4;
	tylocalAGV.In.bUISOTMagSizeLarge1	:= g_tyUIOut.bSOTMagSLarge1;
	tylocalAGV.In.bUISOTMagSizeLarge2	:= g_tyUIOut.bSOTMagSLarge2;
	tylocalAGV.In.bUISOTMagSizeLarge3 := g_tyUIOut.bSOTMagSLarge3;
	//		tylocalAGV.In.bSOTMagSizeLarge4	:= g_tyUIOut.bSOTMagSLarge4;

	tylocalAGV.In.bUIRequestToBring1 := g_tyUIOut.bAIVReqBring1;
	tylocalAGV.In.bUIRequestToBring2 := g_tyUIOut.bAIVReqBring2;
	tylocalAGV.In.bUIRequestToBring3 := g_tyUIOut.bAIVReqBring3;

	tylocalAGV.In.bUIRequestToGet1 := g_tyUIOut.bAIVReqGet1;
	tylocalAGV.In.bUIRequestToGet2 := g_tyUIOut.bAIVReqGet2;
	tylocalAGV.In.bUIRequestToGet3 := g_tyUIOut.bAIVReqGet3;

	tylocalAGV.In.eAGVComProtocol := g_tyMcParamCurr.eAGVComProtocol;

	tylocalAGV.In.bSOTMagReady1 := g_tyUSSOT1.bUSB;
	tylocalAGV.In.bSOTMagReady2 := g_tyUSSOT2.bUSB;
	tylocalAGV.In.bSOTMagReady3 := g_tyUSSOT3.bUSB;

	tylocalAGV.In.bSOTMagError1 := g_tyAlm.bErr;
	tylocalAGV.In.bSOTMagError2 := g_tyAlm.bErr;
	tylocalAGV.In.bSOTMagError3 := g_tyAlm.bErr;

	tylocalAGV.In.bSOTMagAvailable1 := g_tyDSSOT1.bDBA;
	tylocalAGV.In.bSOTMagAvailable2 := g_tyDSSOT2.bDBA;
	tylocalAGV.In.bSOTMagAvailable3 := g_tyDSSOT3.bDBA;

	tylocalAGV.In.bSOTMagSizeLarge1 := g_tyDSSOT1.bDSMagSizeLarge;
	tylocalAGV.In.bSOTMagSizeLarge2 := g_tyDSSOT2.bDSMagSizeLarge;
	tylocalAGV.In.bSOTMagSizeLarge3 := g_tyDSSOT3.bDSMagSizeLarge;

	tylocalAGV.In.bRequestToGet1 := g_tyDSSOT1.bDBA;
	tylocalAGV.In.bRequestToGet2 := g_tyDSSOT2.bDBA;
	tylocalAGV.In.bRequestToGet3 := g_tyDSSOT3.bDBA;
	tylocalAGV.In.bRequestToBring1 := g_tyBuffer1.bMagRemoved;
	tylocalAGV.In.bRequestToBring2 := g_tyBuffer2.bMagRemoved;
	tylocalAGV.In.bRequestToBring3 := g_tyBuffer3.bMagRemoved;

	tylocalAGV.In.bDisableFMWarning := g_tyMcParamCurr.bDisableFMWarning;

	//For Siemen + We fab
	tylocalAGV.In.eCustomerReq := g_tyNtParamCurr.eCustomerReq;

	tylocalAGV.In.bOpsMagConvUL1ReadRFID := g_tyOpsMagConvUL1.bReadRFID;
	tylocalAGV.In.bOpsMagConvUL1WriteRFID := g_tyOpsMagConvUL1.bWriteRFID;

	tylocalAGV.In.bOpsMagConvUL2ReadRFID := g_tyOpsMagConvUL2.bReadRFID;
	tylocalAGV.In.bOpsMagConvUL2WriteRFID := g_tyOpsMagConvUL2.bWriteRFID;

	tylocalAGV.In.bOpsMagConvUL3ReadRFID := g_tyOpsMagConvUL3.bReadRFID;
	tylocalAGV.In.bOpsMagConvUL3WriteRFID := g_tyOpsMagConvUL3.bWriteRFID;

	tylocalAGV.Out.tyDTMagToAGV.bEStopErr  := (tylocalAGV.In.bLinkCoverSWSig = FALSE) OR (tylocalAGV.In.bLinkSafetyRlySig = FALSE);
	(* Always Change If Project Change *)
END_ACTION
```

#### Act_OutputConfig.st - Change By Project
```iecst
ACTION Act_OutputConfig:

	g_tyAGV := tylocalAGV.Out; // Change the Global Naming According to the Physical Hardware Module

END_ACTION
```

#### Cyclic.st - Do Not Change!!!
```iecst
(** 2019-01-11 **)
PROGRAM _CYCLIC

	IF bInitialDone = FALSE THEN
		IF g_tyStartUp.bNtSettingsLoadDone = TRUE THEN
			bInitialDone	:= TRUE;
			Act_Initial;
		END_IF
	ELSE
		Act_InputConfig;
		IF (tylocalAGV.In.bPrep = TRUE) AND (tylocalAGV.In.bEn = TRUE) AND (tylocalAGV.In.bDis = FALSE) THEN

			Act_Background;
			Act_Main;
		ELSE
			IF tylocalAGV.Out.eStat <> AGVMagActIdle THEN
				tylocalAGV.Out.eStatus	:= Done;
			ELSE
				tylocalAGV.Out.eStatus	:= Idle;
			END_IF
		END_IF
		Act_OutputConfig;
		Act_Alarm;
	END_IF

END_PROGRAM
```

#### Act_Initial.st - Do Not Change!!!
```iecst
(** 2019-01-12 **)
ACTION Act_Initial:

	//Initial
	tylocalAGV.Out.sStatTxt	:= a_sStatText[eStat];
	sProgNm	:= 'AGV';
END_ACTION
```

#### Act_Main.st - Do Not Change!!!
```iecst
(** 2019-01-20 **)
ACTION Act_Main:

	tylocalAGV.Out.tyTagToMes.sMachineName := tylocalAGV.In.sJobNo;
	tylocalAGV.Out.tyTagToMes.bError := tylocalAGV.In.bLinkError;
	tylocalAGV.Out.tyTagToMes.bWarning := tylocalAGV.In.bLinkAlarmWarning OR tylocalAGV.In.bLinkAlarmInfo;

	tylocalAGV.Out.bFleetManagerActive := tylocalAGV.In.bDIFleetManagerActive;

	CASE tylocalAGV.In.eAGVComProtocol OF
		McSetAGVCommOPCUA, McSetAGVCommHardIO:
			fbFMOnTimeout(IN:= tylocalAGV.Out.bFleetManagerActive);
			fbFMOffTimeout(IN:= tylocalAGV.Out.bFleetManagerActive = FALSE);
			IF fbFMOnTimeout.Q OR fbFMOffTimeout.Q THEN
				IF tylocalAGV.In.bDisableFMWarning = FALSE THEN
					udiStatus1 := 10006;
				ELSE
					udiStatus1 := 0;
				END_IF
			ELSE
				udiStatus1 := 0;
			END_IF
		McSetAGVCommDisabled:
			udiStatus1 := 0;
	END_CASE

	CASE tylocalAGV.In.eLinkULMag OF
		ULMagDual:
			tylocalAGV.Out.tyTagToMes.nNumberOfPlatforms:= 2;

		ULMagTriple:
			tylocalAGV.Out.tyTagToMes.nNumberOfPlatforms:= 3;

		ULMagQuadruple:
			tylocalAGV.Out.tyTagToMes.nNumberOfPlatforms:= 4;
	END_CASE

	//Online Pulse Status- 500ms Pulse
	fbConnectionAGVTm(IN:= tylocalAGV.Out.tyTagToMes.bActive = FALSE);
	IF fbConnectionAGVTm.Q THEN
		tylocalAGV.Out.tyTagToMes.bActive := TRUE;
	END_IF

	fbConnectionAGVTm1(IN:= tylocalAGV.Out.tyTagToMes.bActive);
	IF fbConnectionAGVTm1.Q THEN
		tylocalAGV.Out.tyTagToMes.bActive := FALSE;
	END_IF

	//Simulation from HMI
	IF tylocalAGV.In.bUIAGVSimulationOn THEN
		bAGVOnline := tylocalAGV.In.bUIAGVOnline;

		tylocalAGV.Out.tyAGVToDTMag.bVEHAuto := tylocalAGV.In.tyUIAGVToDTMagSimulateData.bVEHAuto;
		tylocalAGV.Out.tyAGVToDTMag.bVEHInPos1 := tylocalAGV.In.tyUIAGVToDTMagSimulateData.bVEHInPos1;
		tylocalAGV.Out.tyAGVToDTMag.bVEHInPos2 := tylocalAGV.In.tyUIAGVToDTMagSimulateData.bVEHInPos2;
		tylocalAGV.Out.tyAGVToDTMag.bVEHInPos3 := tylocalAGV.In.tyUIAGVToDTMagSimulateData.bVEHInPos3;
		tylocalAGV.Out.tyAGVToDTMag.bVEH1Occupied := tylocalAGV.In.tyUIAGVToDTMagSimulateData.bVEH1Occupied;
		tylocalAGV.Out.tyAGVToDTMag.bVEH2Occupied := tylocalAGV.In.tyUIAGVToDTMagSimulateData.bVEH2Occupied;
		tylocalAGV.Out.tyAGVToDTMag.bVEH3Occupied := tylocalAGV.In.tyUIAGVToDTMagSimulateData.bVEH3Occupied;
		tylocalAGV.Out.bInternalAGVSimulateOn := TRUE;

	END_IF

	IF EDGEPOS( tylocalAGV.In.bUIAGVSimulationOn = FALSE) THEN
		bAGVOnline := FALSE;

		tylocalAGV.Out.tyAGVToDTMag.bVEHAuto := FALSE;
		tylocalAGV.Out.tyAGVToDTMag.bVEHInPos1 := FALSE;
		tylocalAGV.Out.tyAGVToDTMag.bVEHInPos2 := FALSE;
		tylocalAGV.Out.tyAGVToDTMag.bVEHInPos3 := FALSE;
		tylocalAGV.Out.tyAGVToDTMag.bVEH1Occupied := FALSE;
		tylocalAGV.Out.tyAGVToDTMag.bVEH2Occupied := FALSE;
		tylocalAGV.Out.tyAGVToDTMag.bVEH3Occupied := FALSE;
		tylocalAGV.Out.bInternalAGVSimulateOn := FALSE;

	END_IF

	IF tylocalAGV.In.bOpsRun AND tylocalAGV.In.eLinkAGVComProtocol = McSetAGVCommOPCUA THEN
		tylocalAGV.Out.bInternalAGVOnline := TRUE;
		tylocalAGV.Out.tyTagToMes.bAuto_Run := TRUE;
		//Magazine Conveyor 1
		tylocalAGV.Out.tyDTMagToAGV.bCI1Auto					:= tylocalAGV.In.tyDTMagToAGV1.bCI1Auto;
		tylocalAGV.Out.tyDTMagToAGV.bCI1Rdy  					:= tylocalAGV.In.tyDTMagToAGV1.bCI1Rdy;
		tylocalAGV.Out.tyDTMagToAGV.bCI1MagazineFull			:= tylocalAGV.In.tyDTMagToAGV1.bCI1MagazineFull;
		tylocalAGV.Out.tyDTMagToAGV.bCI1Occupied				:= tylocalAGV.In.tyDTMagToAGV1.bCI1Occupied;
		tylocalAGV.Out.tyDTMagToAGV.bCI1Running				:= tylocalAGV.In.tyDTMagToAGV1.bCI1Running;
		tylocalAGV.Out.tyDTMagToAGV.bCI1IncorrectMagazineModel	:= tylocalAGV.In.bIncorrectMagazine1;

		tylocalAGV.Out.tyTagToMes.tyTagStatOfPlatforms[1].bReqAIVToBring	:= tylocalAGV.In.bRequestToBring1;
		tylocalAGV.Out.tyTagToMes.tyTagStatOfPlatforms[1].bReqAIVToGet		:= tylocalAGV.In.bRequestToGet1;
		tylocalAGV.Out.tyTagToMes.tyTagStatOfPlatforms[1].bError			:= tylocalAGV.In.bSOTMagError1;
		tylocalAGV.Out.tyTagToMes.tyTagStatOfPlatforms[1].bSizeLarge		:= tylocalAGV.In.bSOTMagSizeLarge1;
		tylocalAGV.Out.tyTagToMes.tyTagStatOfPlatforms[1].bReady			:= tylocalAGV.In.bSOTMagReady1;
		tylocalAGV.Out.tyTagToMes.tyTagStatOfPlatforms[1].bAvailable		:= tylocalAGV.In.bSOTMagAvailable1;

		//Magazine Conveyor 2
		tylocalAGV.Out.tyDTMagToAGV.bCI2Auto					:= tylocalAGV.In.tyDTMagToAGV2.bCI2Auto;
		tylocalAGV.Out.tyDTMagToAGV.bCI2Rdy  					:= tylocalAGV.In.tyDTMagToAGV2.bCI2Rdy;
		tylocalAGV.Out.tyDTMagToAGV.bCI2MagazineFull			:= tylocalAGV.In.tyDTMagToAGV2.bCI2MagazineFull;
		tylocalAGV.Out.tyDTMagToAGV.bCI2Occupied				:= tylocalAGV.In.tyDTMagToAGV2.bCI2Occupied;
		tylocalAGV.Out.tyDTMagToAGV.bCI2Running				:= tylocalAGV.In.tyDTMagToAGV2.bCI2Running;
		tylocalAGV.Out.tyDTMagToAGV.bCI2IncorrectMagazineModel	:= tylocalAGV.In.bIncorrectMagazine2;

		tylocalAGV.Out.tyTagToMes.tyTagStatOfPlatforms[2].bReqAIVToBring	:= tylocalAGV.In.bRequestToBring2;
		tylocalAGV.Out.tyTagToMes.tyTagStatOfPlatforms[2].bReqAIVToGet		:= tylocalAGV.In.bRequestToGet2;
		tylocalAGV.Out.tyTagToMes.tyTagStatOfPlatforms[2].bError			:= tylocalAGV.In.bSOTMagError2;
		tylocalAGV.Out.tyTagToMes.tyTagStatOfPlatforms[2].bSizeLarge		:= tylocalAGV.In.bSOTMagSizeLarge2;
		tylocalAGV.Out.tyTagToMes.tyTagStatOfPlatforms[2].bReady			:= tylocalAGV.In.bSOTMagReady2;
		tylocalAGV.Out.tyTagToMes.tyTagStatOfPlatforms[2].bAvailable		:= tylocalAGV.In.bSOTMagAvailable2;

		//Magazine Conveyor 3
		tylocalAGV.Out.tyDTMagToAGV.bCI3Auto					:= tylocalAGV.In.tyDTMagToAGV3.bCI3Auto;
		tylocalAGV.Out.tyDTMagToAGV.bCI3Rdy  					:= tylocalAGV.In.tyDTMagToAGV3.bCI3Rdy;
		tylocalAGV.Out.tyDTMagToAGV.bCI3MagazineFull			:= tylocalAGV.In.tyDTMagToAGV3.bCI3MagazineFull;
		tylocalAGV.Out.tyDTMagToAGV.bCI3Occupied				:= tylocalAGV.In.tyDTMagToAGV3.bCI3Occupied;
		tylocalAGV.Out.tyDTMagToAGV.bCI3Running				:= tylocalAGV.In.tyDTMagToAGV3.bCI3Running;
		tylocalAGV.Out.tyDTMagToAGV.bCI3IncorrectMagazineModel	:= tylocalAGV.In.bIncorrectMagazine3;

		tylocalAGV.Out.tyTagToMes.tyTagStatOfPlatforms[3].bReqAIVToBring	:= tylocalAGV.In.bRequestToBring3;
		tylocalAGV.Out.tyTagToMes.tyTagStatOfPlatforms[3].bReqAIVToGet		:= tylocalAGV.In.bRequestToGet3;
		tylocalAGV.Out.tyTagToMes.tyTagStatOfPlatforms[3].bError			:= tylocalAGV.In.bSOTMagError3;
		tylocalAGV.Out.tyTagToMes.tyTagStatOfPlatforms[3].bSizeLarge		:= tylocalAGV.In.bSOTMagSizeLarge3;
		tylocalAGV.Out.tyTagToMes.tyTagStatOfPlatforms[3].bReady			:= tylocalAGV.In.bSOTMagReady3;
		tylocalAGV.Out.tyTagToMes.tyTagStatOfPlatforms[3].bAvailable		:= tylocalAGV.In.bSOTMagAvailable3;

		//To AGV Side to Check Machine On
		tylocalAGV.Out.bMachineOnline := TRUE;

		//Siemens + Wefabricate
		CASE tylocalAGV.In.eCustomerReq OF
			 Siemens:
				tylocalAGV.Out.tyTagToMes.tyTagStatOfPlatforms[1].bReadRFID 	:= tylocalAGV.In.bOpsMagConvUL1ReadRFID;
				tylocalAGV.Out.tyTagToMes.tyTagStatOfPlatforms[2].bReadRFID 	:= tylocalAGV.In.bOpsMagConvUL2ReadRFID;
				tylocalAGV.Out.tyTagToMes.tyTagStatOfPlatforms[3].bReadRFID 	:= tylocalAGV.In.bOpsMagConvUL3ReadRFID;
				tylocalAGV.Out.tyTagToMes.tyTagStatOfPlatforms[1].bWriteRFID 	:= tylocalAGV.In.bOpsMagConvUL1WriteRFID;
				tylocalAGV.Out.tyTagToMes.tyTagStatOfPlatforms[2].bWriteRFID 	:= tylocalAGV.In.bOpsMagConvUL2WriteRFID;
				tylocalAGV.Out.tyTagToMes.tyTagStatOfPlatforms[3].bWriteRFID 	:= tylocalAGV.In.bOpsMagConvUL3WriteRFID;
			We_Fabricate:
				tylocalAGV.Out.tyTagToMes.tyTagStatOfPlatforms[1].bMagLoaded 	:= tylocalAGV.In.bOpsMagConvUL1ReadRFID;
				tylocalAGV.Out.tyTagToMes.tyTagStatOfPlatforms[2].bMagLoaded 	:= tylocalAGV.In.bOpsMagConvUL2ReadRFID;
				tylocalAGV.Out.tyTagToMes.tyTagStatOfPlatforms[3].bMagLoaded 	:= tylocalAGV.In.bOpsMagConvUL3ReadRFID;
		END_CASE

	ELSE
		tylocalAGV.Out.bInternalAGVOnline := FALSE;
		tylocalAGV.Out.tyTagToMes.bAuto_Run := FALSE;
		//Magazine Conveyor 1
		tylocalAGV.Out.tyDTMagToAGV.bCI1Auto					:= FALSE;
		tylocalAGV.Out.tyDTMagToAGV.bCI1Rdy  					:= FALSE;
		tylocalAGV.Out.tyDTMagToAGV.bCI1Running				:= FALSE;

		//Magazine Conveyor 2
		tylocalAGV.Out.tyDTMagToAGV.bCI2Auto					:= FALSE;
		tylocalAGV.Out.tyDTMagToAGV.bCI2Rdy  					:= FALSE;
		tylocalAGV.Out.tyDTMagToAGV.bCI2Running				:= FALSE;

		//Magazine Conveyor 3
		tylocalAGV.Out.tyDTMagToAGV.bCI3Auto					:= FALSE;
		tylocalAGV.Out.tyDTMagToAGV.bCI3Rdy  					:= FALSE;
		tylocalAGV.Out.tyDTMagToAGV.bCI3Running				:= FALSE;

		tylocalAGV.Out.bMachineOnline := FALSE;

		//Siemens
		tylocalAGV.Out.tyTagToMes.tyTagStatOfPlatforms[1].bReadRFID 	:= FALSE;
		tylocalAGV.Out.tyTagToMes.tyTagStatOfPlatforms[1].bWriteRFID 	:= FALSE;
		tylocalAGV.Out.tyTagToMes.tyTagStatOfPlatforms[2].bReadRFID 	:= FALSE;
		tylocalAGV.Out.tyTagToMes.tyTagStatOfPlatforms[2].bWriteRFID 	:= FALSE;
		tylocalAGV.Out.tyTagToMes.tyTagStatOfPlatforms[3].bReadRFID 	:= FALSE;
		tylocalAGV.Out.tyTagToMes.tyTagStatOfPlatforms[3].bWriteRFID 	:= FALSE;

		IF tylocalAGV.In.bManual THEN

			tylocalAGV.Out.tyTagToMes.tyTagStatOfPlatforms[1].bReqAIVToBring	:= tylocalAGV.In.bUIRequestToBring1;
			tylocalAGV.Out.tyTagToMes.tyTagStatOfPlatforms[1].bReqAIVToGet		:= tylocalAGV.In.bUIRequestToGet1;
			tylocalAGV.Out.tyTagToMes.tyTagStatOfPlatforms[1].bError			:= tylocalAGV.In.bUISOTMagError1;
			tylocalAGV.Out.tyTagToMes.tyTagStatOfPlatforms[1].bSizeLarge		:= tylocalAGV.In.bUISOTMagSizeLarge1;
			tylocalAGV.Out.tyTagToMes.tyTagStatOfPlatforms[1].bReady			:= tylocalAGV.In.bUISOTMagReady1;
			tylocalAGV.Out.tyTagToMes.tyTagStatOfPlatforms[1].bAvailable		:= tylocalAGV.In.bUISOTMagAvailable1;

			tylocalAGV.Out.tyTagToMes.tyTagStatOfPlatforms[2].bReqAIVToBring	:= tylocalAGV.In.bUIRequestToBring2;
			tylocalAGV.Out.tyTagToMes.tyTagStatOfPlatforms[2].bReqAIVToGet		:= tylocalAGV.In.bUIRequestToGet2;
			tylocalAGV.Out.tyTagToMes.tyTagStatOfPlatforms[2].bError			:= tylocalAGV.In.bUISOTMagError2;
			tylocalAGV.Out.tyTagToMes.tyTagStatOfPlatforms[2].bSizeLarge		:= tylocalAGV.In.bUISOTMagSizeLarge2;
			tylocalAGV.Out.tyTagToMes.tyTagStatOfPlatforms[2].bReady			:= tylocalAGV.In.bUISOTMagReady2;
			tylocalAGV.Out.tyTagToMes.tyTagStatOfPlatforms[2].bAvailable		:= tylocalAGV.In.bUISOTMagAvailable2;

			tylocalAGV.Out.tyTagToMes.tyTagStatOfPlatforms[3].bReqAIVToBring	:= tylocalAGV.In.bUIRequestToBring3;
			tylocalAGV.Out.tyTagToMes.tyTagStatOfPlatforms[3].bReqAIVToGet		:= tylocalAGV.In.bUIRequestToGet3;
			tylocalAGV.Out.tyTagToMes.tyTagStatOfPlatforms[3].bError			:= tylocalAGV.In.bUISOTMagError3;
			tylocalAGV.Out.tyTagToMes.tyTagStatOfPlatforms[3].bSizeLarge		:= tylocalAGV.In.bUISOTMagSizeLarge3;
			tylocalAGV.Out.tyTagToMes.tyTagStatOfPlatforms[3].bReady			:= tylocalAGV.In.bUISOTMagReady3;
			tylocalAGV.Out.tyTagToMes.tyTagStatOfPlatforms[3].bAvailable		:= tylocalAGV.In.bUISOTMagAvailable3;

		ELSE

			tylocalAGV.Out.tyTagToMes.tyTagStatOfPlatforms[1].bReqAIVToBring	:= FALSE;
			tylocalAGV.Out.tyTagToMes.tyTagStatOfPlatforms[1].bReqAIVToGet		:= FALSE;
			tylocalAGV.Out.tyTagToMes.tyTagStatOfPlatforms[1].bError			:= FALSE;
			tylocalAGV.Out.tyTagToMes.tyTagStatOfPlatforms[1].bSizeLarge		:= FALSE;
			tylocalAGV.Out.tyTagToMes.tyTagStatOfPlatforms[1].bReady			:= FALSE;
			tylocalAGV.Out.tyTagToMes.tyTagStatOfPlatforms[1].bAvailable		:= FALSE;

			tylocalAGV.Out.tyTagToMes.tyTagStatOfPlatforms[2].bReqAIVToBring	:= FALSE;
			tylocalAGV.Out.tyTagToMes.tyTagStatOfPlatforms[2].bReqAIVToGet		:= FALSE;
			tylocalAGV.Out.tyTagToMes.tyTagStatOfPlatforms[2].bError			:= FALSE;
			tylocalAGV.Out.tyTagToMes.tyTagStatOfPlatforms[2].bSizeLarge		:= FALSE;
			tylocalAGV.Out.tyTagToMes.tyTagStatOfPlatforms[2].bReady			:= FALSE;
			tylocalAGV.Out.tyTagToMes.tyTagStatOfPlatforms[2].bAvailable		:= FALSE;

			tylocalAGV.Out.tyTagToMes.tyTagStatOfPlatforms[3].bReqAIVToBring	:= FALSE;
			tylocalAGV.Out.tyTagToMes.tyTagStatOfPlatforms[3].bReqAIVToGet		:= FALSE;
			tylocalAGV.Out.tyTagToMes.tyTagStatOfPlatforms[3].bError			:= FALSE;
			tylocalAGV.Out.tyTagToMes.tyTagStatOfPlatforms[3].bSizeLarge		:= FALSE;
			tylocalAGV.Out.tyTagToMes.tyTagStatOfPlatforms[3].bReady			:= FALSE;
			tylocalAGV.Out.tyTagToMes.tyTagStatOfPlatforms[3].bAvailable		:= FALSE;

		END_IF

	END_IF

	//first machine
	//connect to ip when feature enable
	//condition: once a mag finished , send data
	//reset counting when unloading new magazine
	//data : send mag Traverser total unload board pulse

	//last machine
	//condition: counting board
	//release non empty magazine with at least more than one board
	//mag  release

END_ACTION
```

#### Act_Alarm.st - Do Not Change!!!
```iecst
(** 2019-03-25 **)
ACTION Act_Alarm:
		//Reset Error
	IF (tylocalAGV.Out.eStatus = Error) AND bRstErr THEN
		//		tylocalAGV.In.eAct	:= AIVMagActIdle;
		//		tylocalAGV.Out.eStat	:= AIVMagActIdle;
	END_IF

	IF tylocalAGV.In.udiRstErr <> udiRstErrOld THEN
		bRstErr			:= TRUE;
		udiRstErrOld	:= tylocalAGV.In.udiRstErr;
	ELSE
		bRstErr			:= FALSE;
	END_IF
	//Error
	IF EDGEPOS(tylocalAGV.Out.eStatus = Error) THEN

		tylocalAGV.Out.tyAlmData.udiCode		:= udiStatus;
		tylocalAGV.Out.tyAlmData.eSeverity		:= AlmSeverityError;
		tylocalAGV.Out.tyAlmData.udiRunTime		:= tylocalAGV.Out.tyAlmData.udiRunTime + 1;
		tylocalAGV.Out.tyAlmData.bAlm			:= TRUE;
		tylocalAGV.Out.tyAlmData.udiModuleNum  	:= udiModuleNum;
		g_tyAlmProgNm.sAGVProgNm				:= tylocalAGV.In.sProgNm;

		tylocalAGV.Out.sStatTxt	:= tylocalAGV.Out.tyAlmData.sAlmMsg;

	ELSIF bRstErr AND (tylocalAGV.Out.tyAlmData.udiCode <> 0) THEN

		tylocalAGV.Out.tyAlmData.udiCode	:= 0;
		tylocalAGV.Out.tyAlmData.eSeverity	:= AlmSeverityNA;
		tylocalAGV.Out.tyAlmData.bAlm			:= FALSE;
		tylocalAGV.Out.sStatTxt	:= a_sStatText[tylocalAGV.Out.eStat];

	END_IF

	//Warning
	tylocalAGV.Out.tyAlmData1.udiCode			:= udiStatus1;
	tylocalAGV.Out.tyAlmData1.eSeverity			:= AlmSeverityWarning;
	tylocalAGV.Out.tyAlmData1.udiRunTime		:= tylocalAGV.Out.tyAlmData1.udiRunTime + 1;
	tylocalAGV.Out.tyAlmData1.bWarning			:= TRUE;
	tylocalAGV.Out.tyAlmData1.udiModuleNum  	:= udiModuleNum;
	g_tyAlmProgNm.sAGVProgNm					:= tylocalAGV.In.sProgNm;

END_ACTION
```

#### Local.var - Do Not Change!!!
```iecst
(*2019-01-20*)
VAR
	tylocalAGV : tyAGVCom;
END_VAR
(**)
(*Local Action, State & Status*)
VAR
	eAct : eAGVMagAction := AGVMagActIdle;
	eStat : eAGVMagAction := AGVMagActIdle;
	eStatus : eFBStatus := Idle;
	eStatus1 : eFBStatus := Idle;
	udiStatus : UDINT := 0;
	udiStatus1 : UDINT := 0;
	sStatTxt : STRING[100] := '';
	a_sStatText : ARRAY[0..50] OF STRING[100] := ['Idling','AIV Magazine Ready Enter And Communicating AIV','AIV Magazine Ready Exit And Communicating AIV',48('')];
END_VAR
(**)
(*Local Alarm*)
VAR
	tyAlmData : tyAlmDat;
	tyAlmData1 : tyAlmDat;
	a_tyAlmText : ARRAY[10000..10099] OF tyAlmTxt := [(sAlmText:='Magazine Is Present Before Entering',sRcyText:='Remove Magazine To Continue Operation.'),(sAlmText:='AIV Not In Enter Position',sRcyText:='Adjust AIV Position And Restart Operation.'),(sAlmText:='Transfer In Time Out While Transporting',sRcyText:='Adjust Magazine Position Or Transporting Time.'),(sAlmText:='Magazine Is Not Present Before Exiting',sRcyText:='Magazine Has Taken Away, Restart Operation.'),(sAlmText:='AIV Not In Exit Position',sRcyText:='Adjust AIV Position And Restart Operation.'),(sAlmText:='Transfer Out Time Out While Transporting',sRcyText:='Adjust Magazine Position Or Transporting Time.'),(sAlmText:='Fleet Manager Is Offline',sRcyText:='Please check the connectivity signal to Fleetmanger'),93((0))];
END_VAR
(**)
(*Local Output*)
VAR
	bMcRunRdy : BOOL;
	bRdyEnt : BOOL;
	bRdyExit : BOOL;
	bMag1Ent : BOOL;
	bMag1Exit : BOOL;
END_VAR
(**)
(*Local Input*)
VAR
	udiRstErr : UDINT := 0;
	bPrep : BOOL := TRUE;
	bEn : BOOL := TRUE;
	bDis : BOOL := FALSE;
	bNtSettingsLoadDone : BOOL := TRUE;
	tyAGVToDTMag : tyTagAGVToDTMag;
	tyDTMagToAGV : tyTagDTMagToAGV;
	bAGVOnline : BOOL;
	bMachineOnline : BOOL;
	bInternalAGVOnline : BOOL;
	bInternalAGVSimulateOn : BOOL;
	tyDTMagToAGV1 : tyTagDTMagToAGV;
	tyDTMagToAGV2 : tyTagDTMagToAGV;
	tyDTMagToAGV3 : tyTagDTMagToAGV;
	bRequestToBring1 : BOOL;
	bRequestToGet1 : BOOL;
	bRequestToBring2 : BOOL;
	bRequestToGet2 : BOOL;
	bRequestToBring3 : BOOL;
	bRequestToGet3 : BOOL;
	bRequestToBring4 : BOOL;
	bRequestToGet4 : BOOL;
END_VAR
(**)
(*Local*)
VAR
	bRstErr : BOOL;
	udiRstErrOld : UDINT;
	bInitDone : BOOL;
	bInitialDone : BOOL;
	bFleetManagerActive : BOOL;
	fbFMOnTimeout : TON := (PT:=T#20s);
	fbFMOffTimeout : TON := (PT:=T#20s);
	usiStep : USINT;
	eStatOld : eAGVMagAction := AGVMagActIdle;
	fbConnectionTmCCS : TON := (PT:=T#250ms);
	fbConnectionAGVTm : TON := (PT:=T#500ms);
	fbConnectionAGVTm1 : TON := (PT:=T#500ms);
END_VAR
(**)
VAR
	udiModuleNum : UDINT := 6111;
END_VAR
(*AGV Batch Count*)
VAR
	tyTagFromLoader : tyStatFromLoader;
END_VAR
```

#### InputRef.var - not listed in the package file held
```iecst
(*2019-01-20*)
(**)
(*General*)
VAR
	p_udiRstErr : REFERENCE TO UDINT;
	p_bPrep : REFERENCE TO BOOL;
	p_bEn : REFERENCE TO BOOL;
	p_bDis : REFERENCE TO BOOL;
END_VAR
(**)
(*Configuration*)
VAR
	p_sProgNm : REFERENCE TO STRING[15];
	p_bNtSettingsLoadDone : REFERENCE TO BOOL;
	p_sJobNo : REFERENCE TO STRING[30];
END_VAR
(**)
(*Input*)
VAR
	p_bManual : REFERENCE TO BOOL;
	p_tyDTMagToAGV1 : REFERENCE TO tyTagDTMagToAGV;
	p_tyDTMagToAGV2 : REFERENCE TO tyTagDTMagToAGV;
	p_tyDTMagToAGV3 : REFERENCE TO tyTagDTMagToAGV;
	p_bOpsRun : REFERENCE TO BOOL;
	p_bLinkOpsSimu : REFERENCE TO BOOL;
	p_bIncorrectMagazine1 : REFERENCE TO BOOL;
	p_bIncorrectMagazine2 : REFERENCE TO BOOL;
	p_bIncorrectMagazine3 : REFERENCE TO BOOL;
END_VAR
(*Simulate Data*)
VAR
	p_tyUIAGVToDTMagSimulateData : REFERENCE TO tyTagAGVToDTMag;
	p_bUIAGVOnline : REFERENCE TO BOOL;
	p_bUIAGVSimulationOn : REFERENCE TO BOOL;
	p_bAGVRdyEnter1 : REFERENCE TO BOOL;
	p_bAGVRdyExit1 : REFERENCE TO BOOL;
	p_bAGVRdyEnter2 : REFERENCE TO BOOL;
	p_bAGVRdyExit2 : REFERENCE TO BOOL;
	p_bAGVRdyEnter3 : REFERENCE TO BOOL;
	p_bAGVRdyExit3 : REFERENCE TO BOOL;
END_VAR
(**)
VAR
	p_bRequestToBring1 : REFERENCE TO BOOL;
	p_bRequestToBring2 : REFERENCE TO BOOL;
	p_bRequestToBring3 : REFERENCE TO BOOL;
	p_bRequestToBring4 : REFERENCE TO BOOL;
	p_bRequestToGet1 : REFERENCE TO BOOL;
	p_bRequestToGet2 : REFERENCE TO BOOL;
	p_bRequestToGet3 : REFERENCE TO BOOL;
	p_bRequestToGet4 : REFERENCE TO BOOL;
	p_bUISOTMagError1 : REFERENCE TO BOOL;
	p_bUISOTMagError2 : REFERENCE TO BOOL;
	p_bUISOTMagError3 : REFERENCE TO BOOL;
	p_bUISOTMagReady1 : REFERENCE TO BOOL;
	p_bUISOTMagReady2 : REFERENCE TO BOOL;
	p_bUISOTMagReady3 : REFERENCE TO BOOL;
	p_bUISOTMagAvailable1 : REFERENCE TO BOOL;
	p_bUISOTMagAvailable2 : REFERENCE TO BOOL;
	p_bUISOTMagAvailable3 : REFERENCE TO BOOL;
	p_bUISOTMagSizeLarge1 : REFERENCE TO BOOL;
	p_bUISOTMagSizeLarge2 : REFERENCE TO BOOL;
	p_bUISOTMagSizeLarge3 : REFERENCE TO BOOL;
	p_bUIRequestToBring1 : REFERENCE TO BOOL;
	p_bUIRequestToBring2 : REFERENCE TO BOOL;
	p_bUIRequestToBring3 : REFERENCE TO BOOL;
	p_bUIRequestToGet1 : REFERENCE TO BOOL;
	p_bUIRequestToGet2 : REFERENCE TO BOOL;
	p_bUIRequestToGet3 : REFERENCE TO BOOL;
	p_bDIFleetManagerActive : REFERENCE TO BOOL;
	p_eAGVComProtocol : REFERENCE TO eMcAGVCommProtocol;
	p_bSOTMagError1 : REFERENCE TO BOOL;
	p_bSOTMagSizeLarge1 : REFERENCE TO BOOL;
	p_bSOTMagReady1 : REFERENCE TO BOOL;
	p_bSOTMagAvailable1 : REFERENCE TO BOOL;
	p_bSOTMagError2 : REFERENCE TO BOOL;
	p_bSOTMagSizeLarge2 : REFERENCE TO BOOL;
	p_bSOTMagReady2 : REFERENCE TO BOOL;
	p_bSOTMagAvailable2 : REFERENCE TO BOOL;
	p_bSOTMagError3 : REFERENCE TO BOOL;
	p_bSOTMagSizeLarge3 : REFERENCE TO BOOL;
	p_bSOTMagReady3 : REFERENCE TO BOOL;
	p_bSOTMagAvailable3 : REFERENCE TO BOOL;
	p_bDisableFMWarning : REFERENCE TO BOOL;
END_VAR
(*Simens*)
VAR
	p_eCustomerReq : REFERENCE TO eCustomer;
	p_bOpsMagConvUL1ReadRFID : REFERENCE TO BOOL;
	p_bOpsMagConvUL1WriteRFID : REFERENCE TO BOOL;
	p_bOpsMagConvUL2ReadRFID : REFERENCE TO BOOL;
	p_bOpsMagConvUL2WriteRFID : REFERENCE TO BOOL;
	p_bOpsMagConvUL3ReadRFID : REFERENCE TO BOOL;
	p_bOpsMagConvUL3WriteRFID : REFERENCE TO BOOL;
END_VAR
```

#### InputRef_Link.var - not listed in the package file held
```iecst
(*2018-12-08*)
(**)
(*External Data*)
(**)
VAR
	p_bLinkCoverSWSig : REFERENCE TO BOOL;
	p_bLinkSafetyRlySig : REFERENCE TO BOOL;
	p_bLinkAlarmWarning : REFERENCE TO BOOL;
	p_bLinkAlarmInfo : REFERENCE TO BOOL;
	p_bLinkError : REFERENCE TO BOOL;
	p_eLinkULMag : REFERENCE TO eULMag;
	p_eLinkAGVComProtocol : REFERENCE TO eMcAGVCommProtocol;
END_VAR
```

#### Act_Action.st - not listed in the package file held
```iecst
(** 2019-01-09 **)
ACTION Act_Action:

	//Reset Error
	IF (eStatus = Error) AND bRstErr THEN
//		p_eAct	:= AIVMagActIdle;
//		eStat	:= AIVMagActIdle;
	END_IF

	//Set p_eAct
	IF eStatus = Idle OR eStatus = Busy OR eStatus = Done THEN
//		eStat	:= p_eAct;
	END_IF

END_ACTION
```

#### Act_Alarm1.st - not listed in the package file held
```iecst
(** 2019-03-25 **)
ACTION Act_Alarm1:

	//Warning
	tyAlmData1.sProgNm		:= p_sProgNm;
	tyAlmData1.udiCode		:= udiStatus1;
	tyAlmData1.eSeverity	:= AlmSeverityWarning;
	tyAlmData1.udiRunTime	:= tyAlmData1.udiRunTime + 1;
	tyAlmData1.bWarning			:= TRUE;
	tyAlmData1.udiModuleNum  := udiModuleNum;
	g_sAGVComProgNm		:= p_sProgNm;
	//Get Error Message
	IF tyAlmData1.udiCode < 10000 OR tyAlmData1.udiCode > 10099 THEN
		tyAlmData1.sAlmMsg	:= 'Unknown';
		tyAlmData1.sRcyMsg	:= 'Unknown';
	ELSE
		tyAlmData1.sAlmMsg	:= a_tyAlmText[tyAlmData1.udiCode].sAlmText;
		tyAlmData1.sRcyMsg	:= a_tyAlmText[tyAlmData1.udiCode].sRcyText;
	END_IF

END_ACTION
```

#### Act_InitGlobal.st - not listed in the package file held
```iecst
(** 2018-12-08 **)
ACTION Act_InitGlobal:

	(* Always Change If Project Change *)

	//Pass Data To Link
	p_bLinkSafetyRlySig ACCESS p_DISafetyRlySig;
	p_bLinkCoverSWSig ACCESS p_DICoverSWSig;
	p_bLinkAlarmWarning ACCESS p_AlarmWarning;
	p_bLinkAlarmInfo ACCESS p_AlarmInfo;
	p_bLinkError ACCESS p_AlarmErr;
	p_eLinkULMag ACCESS p_NtParamProjMag;
	p_eLinkAGVComProtocol ACCESS p_McParamAGVComProtocol;

	//Pass Data To Internal Use
	p_bOpsRun ACCESS p_OpsRun;
	p_bManual ACCESS p_UIUIMnlMod;
	p_bPrep ACCESS p_NtParamProjAGVPrep;
	p_tyDTMagToAGV1 ACCESS p_AGVMag1DTMagToAGV;
	p_tyDTMagToAGV2 ACCESS p_AGVMag2DTMagToAGV;
	p_tyDTMagToAGV3 ACCESS p_AGVMag3DTMagToAGV;
	p_udiRstErr	ACCESS p_RstErrReset;
	p_sProgNm ACCESS p_NtParamAGVProgNm;
	p_bNtSettingsLoadDone ACCESS p_StartupNtSettingsLoadDone;
	p_bIncorrectMagazine1 ACCESS p_OpsMagConvUL1IncorrectMagModel;
	p_bIncorrectMagazine2 ACCESS p_OpsMagConvUL2IncorrectMagModel;
	p_bIncorrectMagazine3 ACCESS p_OpsMagConvUL3IncorrectMagModel;

	p_tyUIAGVToDTMagSimulateData ACCESS p_UIAGVSimulateSig;
	p_bUIAGVOnline ACCESS p_UIAGVSimulateOnline;
	p_bUIAGVSimulationOn ACCESS p_UIAGVSimulationOn;

	p_sJobNo ACCESS p_NtParamJobNo;

	p_bAGVRdyEnter1 ACCESS p_AGVMag1RdyEnter;
	p_bAGVRdyExit1 ACCESS p_AGVMag1RdyExit;
	p_bAGVRdyEnter2 ACCESS p_AGVMag2RdyEnter;
	p_bAGVRdyExit2 ACCESS p_AGVMag2RdyExit;
	p_bAGVRdyEnter3 ACCESS p_AGVMag3RdyEnter;
	p_bAGVRdyExit3 ACCESS p_AGVMag3RdyExit;

	p_bDIFleetManagerActive ACCESS p_DIFleetManagerActive;

	p_bUISOTMagError1	ACCESS p_UISOTMagErr1;
	p_bUISOTMagError2	ACCESS p_UISOTMagErr2;
	p_bUISOTMagError3	ACCESS p_UISOTMagErr3;
	//		p_bSOTMagError4	ACCESS p_UISOTMagErr4;
	p_bUISOTMagReady1	ACCESS p_UISOTMagRdy1;
	p_bUISOTMagReady2	ACCESS p_UISOTMagRdy2;
	p_bUISOTMagReady3	ACCESS p_UISOTMagRdy3;
	//		p_bSOTMagReady4	ACCESS p_UISOTMagRdy4;
	p_bUISOTMagAvailable1	ACCESS p_UISOTMagAvail1;
	p_bUISOTMagAvailable2	ACCESS p_UISOTMagAvail2;
	p_bUISOTMagAvailable3	ACCESS p_UISOTMagAvail3;
	//		p_bSOTMagAvailable4	ACCESS p_UISOTMagAvail4;
	p_bUISOTMagSizeLarge1	ACCESS p_UISOTMagSLarge1;
	p_bUISOTMagSizeLarge2	ACCESS p_UISOTMagSLarge2;
	p_bUISOTMagSizeLarge3 ACCESS p_UISOTMagSLarge3;
	//		p_bSOTMagSizeLarge4	ACCESS p_UISOTMagSLarge4;

	p_bUIRequestToBring1 ACCESS p_UIAIVReqBring1;
	p_bUIRequestToBring2 ACCESS p_UIAIVReqBring2;
	p_bUIRequestToBring3 ACCESS p_UIAIVReqBring3;

	p_bUIRequestToGet1 ACCESS p_UIAIVReqGet1;
	p_bUIRequestToGet2 ACCESS p_UIAIVReqGet2;
	p_bUIRequestToGet3 ACCESS p_UIAIVReqGet3;

	p_eAGVComProtocol ACCESS p_McParamAGVComProtocol;

	p_bSOTMagReady1 ACCESS p_USSOT1USB;
	p_bSOTMagReady2 ACCESS p_USSOT2USB;
	p_bSOTMagReady3 ACCESS p_USSOT3USB;

	p_bSOTMagError1 ACCESS p_AlarmErr;
	p_bSOTMagError2 ACCESS p_AlarmErr;
	p_bSOTMagError3 ACCESS p_AlarmErr;

	p_bSOTMagAvailable1 ACCESS p_DSSOT1DBA;
	p_bSOTMagAvailable2 ACCESS p_DSSOT2DBA;
	p_bSOTMagAvailable3 ACCESS p_DSSOT3DBA;

	p_bSOTMagSizeLarge1 ACCESS p_DSSOT1MagSizeLarge;
	p_bSOTMagSizeLarge2 ACCESS p_DSSOT2MagSizeLarge;
	p_bSOTMagSizeLarge3 ACCESS p_DSSOT3MagSizeLarge;

	p_bRequestToGet1 ACCESS p_DSSOT1DBA;
	p_bRequestToGet2 ACCESS p_DSSOT2DBA;
	p_bRequestToGet3 ACCESS p_DSSOT3DBA;
	p_bRequestToBring1 ACCESS p_Buffer1MagRemoved;
	p_bRequestToBring2 ACCESS p_Buffer2MagRemoved;
	p_bRequestToBring3 ACCESS p_Buffer3MagRemoved;

	p_bDisableFMWarning ACCESS p_McParamDisableFMWarning;

	//For Siemen + We fab
	p_eCustomerReq ACCESS p_NtParamCustomerReq;

	p_bOpsMagConvUL1ReadRFID ACCESS p_OpsMagConvUL1ReadRFID;
	p_bOpsMagConvUL1WriteRFID ACCESS p_OpsMagConvUL1WriteRFID;

	p_bOpsMagConvUL2ReadRFID ACCESS p_OpsMagConvUL2ReadRFID;
	p_bOpsMagConvUL2WriteRFID ACCESS p_OpsMagConvUL2WriteRFID;

	p_bOpsMagConvUL3ReadRFID ACCESS p_OpsMagConvUL3ReadRFID;
	p_bOpsMagConvUL3WriteRFID ACCESS p_OpsMagConvUL3WriteRFID;

	(* Always Change If Project Change *)
END_ACTION
```

#### Act_InitLocal.st - not listed in the package file held
```iecst
(** 2019-01-20 **)
ACTION Act_InitLocal:

	//Input Reference Link To Local Variable
	p_udiRstErr ACCESS ADR(udiRstErr);
	p_bPrep ACCESS ADR(bPrep);
	p_bEn ACCESS ADR(bEn);
	p_bDis ACCESS ADR(bDis);
	p_sProgNm ACCESS ADR(sProgNm);
	p_bNtSettingsLoadDone ACCESS ADR(bNtSettingsLoadDone);
	p_tyDTMagToAGV1 ACCESS ADR(tyDTMagToAGV1);
	p_tyDTMagToAGV2 ACCESS ADR(tyDTMagToAGV2);
	p_tyDTMagToAGV3 ACCESS ADR(tyDTMagToAGV3);

	p_bRequestToBring1 ACCESS ADR(bRequestToBring1);
	p_bRequestToGet1 ACCESS ADR(bRequestToGet1);
	p_bRequestToBring2 ACCESS ADR(bRequestToBring2);
	p_bRequestToGet2 ACCESS ADR(bRequestToGet2);
	p_bRequestToBring3 ACCESS ADR(bRequestToBring3);
	p_bRequestToGet3 ACCESS ADR(bRequestToGet3);
	p_bRequestToBring4 ACCESS ADR(bRequestToBring4);
	p_bRequestToGet4 ACCESS ADR(bRequestToGet4);

END_ACTION
```

#### Act_Link.st - not listed in the package file held
```iecst
(** 2018-12-08 **)
ACTION Act_Link:

	tyDTMagToAGV.bEStopErr  := (p_bLinkCoverSWSig = FALSE) OR (p_bLinkSafetyRlySig = FALSE);

END_ACTION
```

#### Act_LinkAction.st - not listed in the package file held
```iecst
(** 2019-03-29 **)
ACTION Act_LinkAction:

END_ACTION
```

#### Init.st - not listed in the package file held
```iecst
(** 2019-01-20 **)
PROGRAM _INIT

	(* Always Change If Project Change *)

	sProgNm	:= 'AGV';

	//Physical Configuration

	//Pass Address To Global Address For External Use
	//Action, State & Status
	p_AGVStat		     := ADR(eStat);
	p_AGVStatus		     := ADR(eStatus);
	p_AGVStatTxt	     := ADR(sStatTxt);

	//Alarm
	p_AGVAlmData		 := ADR(tyAlmData);
	p_AGVAlmData1		 := ADR(tyAlmData1);
	//Output
	p_AGVTagAGVToDTMag 	 := ADR(tyAGVToDTMag);
	p_AGVOnline		 	 := ADR(bInternalAGVOnline);
	p_MachineOnline		 := ADR(bMachineOnline);
	p_DTMagToAGV 		 := ADR(tyDTMagToAGV);
	p_AGVSimulationOn 	 := ADR(bInternalAGVSimulateOn);
	p_TagToMes			 := ADR(tyTagToMes);
	p_TagFromMes		 := ADR(tyTagFromMes);
	p_FleetManagerActive := ADR(bFleetManagerActive);

	//For Siemen
	p_TagToMesMagConv1		:= ADR(tyTagToMes.tyTagStatOfPlatforms[1]);
	p_TagToMesMagConv2		:= ADR(tyTagToMes.tyTagStatOfPlatforms[2]);
	p_TagToMesMagConv3		:= ADR(tyTagToMes.tyTagStatOfPlatforms[3]);
	p_TagFromMesMagConv1	:= ADR(tyTagFromMes.tyTagStatOfPlatforms[1]);
	p_TagFromMesMagConv2	:= ADR(tyTagFromMes.tyTagStatOfPlatforms[2]);
	p_TagFromMesMagConv3	:= ADR(tyTagFromMes.tyTagStatOfPlatforms[3]);

	(* Always Change If Project Change *)

END_PROGRAM
```

### Program Logical/AGVCom/AGV1 (IEC) - 1.00.0 - NtSMEMA v5.00.0

#### InputRef.var
```iecst
(*2019-01-20*)
(**)
(*General*)
VAR
	p_eAct : REFERENCE TO eAGVMagAction;
	p_udiRstErr : REFERENCE TO UDINT;
	p_bPrep : REFERENCE TO BOOL;
	p_bEn : REFERENCE TO BOOL;
	p_bDis : REFERENCE TO BOOL;
END_VAR
(**)
(*Configuration*)
VAR
	p_sProgNm : REFERENCE TO STRING[15];
	p_bNtSettingsLoadDone : REFERENCE TO BOOL;
	p_diTxInTimeOut : REFERENCE TO DINT;
	p_diTxOutTimeOut : REFERENCE TO DINT;
	p_eDirection : REFERENCE TO eConvDir;
END_VAR
(**)
(*Input*)
VAR
	p_tyAGVToDTMag : REFERENCE TO tyTagAGVToDTMag;
	p_bBufferMagPresent : REFERENCE TO BOOL;
	p_bMagConvLftSen : REFERENCE TO BOOL;
	p_bMagConvRgtSen : REFERENCE TO BOOL;
	p_bMagConvMtrIn : REFERENCE TO BOOL;
	p_bMagConvMtrOut : REFERENCE TO BOOL;
	p_bNtParamAGVInPosSenPrep : REFERENCE TO BOOL;
	p_bAGVInPosSen1 : REFERENCE TO BOOL;
	p_bAGVInPosSen2 : REFERENCE TO BOOL;
	p_bSOTRcvOk : REFERENCE TO BOOL;
	p_bSOTErr : REFERENCE TO BOOL;
	p_bSOTRdy : REFERENCE TO BOOL;
	p_bSOTAvailable : REFERENCE TO BOOL;
END_VAR
```

#### InputRef_Link.var
```iecst
(*2018-12-08*)
(**)
(*External Data*)
VAR
	p_bLinkAGVOnline : REFERENCE TO BOOL;
	p_bLinkOpsRun : REFERENCE TO BOOL;
END_VAR
(**)
VAR
	p_tyLinkBufferStat : REFERENCE TO tyBffrStat;
	p_tyLinkAGVtoDTMag : REFERENCE TO tyTagAGVToDTMag;
	p_bLinkProjMag1ConvPrep : REFERENCE TO BOOL;
	p_bLinkProjMagConvLane1Prep : REFERENCE TO BOOL;
END_VAR
```

#### Act_Action.st
```iecst
(** 2019-01-09 **)
ACTION Act_Action:

	//Reset Error
	IF (eStatus = Error) AND bRstErr THEN
		p_eAct	:= AGVMagActIdle;
		eStat	:= AGVMagActIdle;
	END_IF

	//Set p_eAct
	IF eStatus = Idle OR eStatus = Busy OR eStatus = Done THEN
		eStat	:= p_eAct;
	END_IF

END_ACTION
```

#### Act_Alarm.st
```iecst
(** 2019-03-25 **)
ACTION Act_Alarm:

	//Error
	IF EDGEPOS(eStatus = Error) THEN

		tyAlmData.sProgNm		:= p_sProgNm;
		tyAlmData.udiCode		:= udiStatus;
		tyAlmData.eSeverity		:= AlmSeverityError;
		tyAlmData.udiRunTime	:= tyAlmData.udiRunTime + 1;
		tyAlmData.bAlm			:= TRUE;
		tyAlmData.udiModuleNum  := udiModuleNum;
		g_sAGVProgNm		:= p_sProgNm;

		//Get Error Message
		IF tyAlmData.udiCode < 10000 OR tyAlmData.udiCode > 10099 THEN
			tyAlmData.sAlmMsg	:= 'Unknown';
			tyAlmData.sRcyMsg	:= 'Unknown';
		ELSE
			tyAlmData.sAlmMsg	:= a_tyAlmText[tyAlmData.udiCode].sAlmText;
			tyAlmData.sRcyMsg	:= a_tyAlmText[tyAlmData.udiCode].sRcyText;
		END_IF

		sStatTxt	:= tyAlmData.sAlmMsg;

	ELSIF bRstErr AND (tyAlmData.udiCode <> 0) THEN

		tyAlmData.udiCode	:= 0;
		tyAlmData.eSeverity	:= AlmSeverityNA;
		tyAlmData.sAlmMsg	:= '';
		tyAlmData.sRcyMsg	:= '';
		tyAlmData.bAlm			:= FALSE;
		sStatTxt	:= a_sStatText[eStat];

	END_IF

END_ACTION
```

#### Act_InitGlobal.st
```iecst
(** 2018-12-08 **)
ACTION Act_InitGlobal:

	(* Always Change If Project Change *)

	//Pass Data To Link
	p_bLinkOpsRun ACCESS p_OpsRun;

	p_tyLinkBufferStat ACCESS p_Buffer1BffrStat;
	p_bLinkAGVOnline ACCESS p_AGVOnline;
	p_tyLinkAGVtoDTMag ACCESS p_AGVTagAGVToDTMag;
	p_bLinkProjMag1ConvPrep ACCESS p_NtParamProjMag1ConvPrep;
	p_bLinkProjMagConvLane1Prep ACCESS p_NtParamProjMagConvLane1Prep;

	//Pass Data To Internal Use
//	p_eAct ACCESS p_OpsMagConvUL1AGVMagAct;
	p_udiRstErr	ACCESS p_RstErrReset;
	p_bPrep ACCESS p_NtParamProjAGVPrep;
	p_sProgNm ACCESS p_NtParamAGVMag1ProgNm;
	p_diTxInTimeOut ACCESS p_McParamMag1ConvRunTmOut;
	p_diTxOutTimeOut ACCESS p_McParamMag1ConvRunTmOut;
	p_eDirection ACCESS p_NtParamProjMagConvDir;
	p_bBufferMagPresent ACCESS p_DIMagPresentSen1;
	p_bMagConvLftSen ACCESS p_DIMagPresentSen1;
	p_bMagConvRgtSen ACCESS p_DIMagConvEntSen1;
	p_bMagConvMtrIn ACCESS p_MagConv2Clp1MtrSigOnOrLToR;
	p_bMagConvMtrOut ACCESS p_MagConv2Clp1MtrDirOrRToL;
	p_bNtSettingsLoadDone ACCESS p_StartupNtSettingsLoadDone;
	p_bAGVInPosSen1	ACCESS p_DIMag1AIVInPosSen1;
	p_bAGVInPosSen2	ACCESS p_DIMag1AIVInPosSen2;
	p_bNtParamAGVInPosSenPrep ACCESS p_NtParamProjAIVInPosSenPrep;
	p_bSOTRcvOk ACCESS p_DISOT1Receive;
	p_bSOTErr ACCESS p_DISOT1Error;
	p_bSOTRdy ACCESS p_DISOT1Ready;
	p_bSOTAvailable ACCESS p_DISOT1Available;
	p_bEn ACCESS p_McParamAGVComEn;

	(* Always Change If Project Change *)

END_ACTION
```

#### Act_Initial.st
```iecst
(** 2019-01-12 **)
ACTION Act_Initial:

	//Initial
	tylocalAGV.Out.sStatTxt	:= a_sStatText[eStat];

	fbTxInTimer(IN := FALSE);
	fbTxOutTimer(IN := FALSE);
	fbMagOutTrig(CLK := FALSE);

	tylocalAGV.Out.bMcRunRdy			:= FALSE;
	tylocalAGV.Out.bRdyEnt			 	:= FALSE;
	tylocalAGV.Out.bRdyExit				:= FALSE;
	tylocalAGV.Out.bMagConvRun	    	:= FALSE;

END_ACTION
```

#### Act_InitLocal.st
```iecst
(** 2019-01-20 **)
ACTION Act_InitLocal:

	//Input Reference Link To Local Variable
	p_eAct ACCESS ADR(eAct);
	p_udiRstErr ACCESS ADR(udiRstErr);
	p_bPrep ACCESS ADR(bPrep);
	p_bEn ACCESS ADR(bEn);
	p_bDis ACCESS ADR(bDis);
	p_sProgNm ACCESS ADR(sProgNm);
	p_tyAGVToDTMag ACCESS ADR(tyAGVToDTMag);
	p_bNtSettingsLoadDone ACCESS ADR(bNtSettingsLoadDone);
	p_diTxInTimeOut ACCESS ADR(diTxInTimeOut);
	p_diTxOutTimeOut ACCESS ADR(diTxOutTimeOut);
	p_eDirection ACCESS ADR(eDirection);
	p_bBufferMagPresent ACCESS ADR(bBufferMagPresent);
	p_bMagConvLftSen ACCESS ADR(bMagConvLftSen);
	p_bMagConvRgtSen ACCESS ADR(bMagConvRgtSen);
	p_bMagConvMtrIn ACCESS ADR(bMagConvMtrIn);
	p_bMagConvMtrOut ACCESS ADR(bMagConvMtrOut);
	p_bAGVInPosSen1	ACCESS ADR(bAGVInPosSen1);
	p_bAGVInPosSen2	ACCESS ADR(bAGVInPosSen2);
	p_bNtParamAGVInPosSenPrep ACCESS ADR(bNtParamAGVInPosSenPrep);
END_ACTION
```

#### Act_InputConfig.st
```iecst
ACTION Act_InputConfig:

	(* Always Change If Project Change *)

	//Pass Data To Link
	tylocalAGV.In.bLinkOpsRun := g_tyOps.bRun;

	tylocalAGV.In.tyLinkBufferStat := g_tyBuffer1.tyBufferStat;
	tylocalAGV.In.bLinkAGVOnline := g_tyAGV.bInternalAGVOnline;
	tylocalAGV.In.tyLinkAGVtoDTMag := g_tyAGV.tyAGVToDTMag;

	//Pass Data To Internal Use
//	tylocalAGV.In.eAct := g_tyOpsMagConvUL1AGVMagAct;
	tylocalAGV.In.udiRstErr	:= g_tyRstErrOut.udiRstErr;
	tylocalAGV.In.bPrep := g_tyNtParamCurr.bProjAGVPrep;
	tylocalAGV.In.sProgNm := g_tyNtParamCurr.sAGVMag1ProgNm;

	tylocalAGV.In.diTxInTimeOut := g_tyMcParam.tMag1ConvRunTmOut;
	tylocalAGV.In.diTxOutTimeOut := g_tyMcParam.tMag1ConvRunTmOut;

	tylocalAGV.In.eDirection := g_tyNtParamCurr.bProjMagConvDir;
	tylocalAGV.In.bBufferMagPresent := g_tyDInput.bMagPresentSen1;
	tylocalAGV.In.bMagConvLftSen := g_tyDInput.bMagPresentSen1;
	tylocalAGV.In.bMagConvRgtSen := g_tyDInput.bMagConvEntSen1;
	tylocalAGV.In.bMagConvMtrIn := g_tyMagConv2Clp1.bMtrSigOnOrLToR;
	tylocalAGV.In.bMagConvMtrOut := g_tyMagConv2Clp1.bMtrDirOrRToL;

	tylocalAGV.In.bAGVInPosSen1	:= g_tyDInput.bMag1AIVInPosSen1;
	tylocalAGV.In.bAGVInPosSen2	:= g_tyDInput.bMag1AIVInPosSen2;

	tylocalAGV.In.bNtParamAGVInPosSenPrep := g_tyNtParamCurr.bProjAIVInPosSenPrep;

	tylocalAGV.In.bSOTRcvOk := g_tyDInput.bSOT1Receive;
	tylocalAGV.In.bSOTErr := g_tyDInput.bSOT1AIVError;
	tylocalAGV.In.bSOTRdy := g_tyDInput.bSOT1AIVReady;
	tylocalAGV.In.bSOTAvailable := g_tyDInput.bSOT1AIVAvailable;
	tylocalAGV.In.bEn := g_tyMcParam.AGVComEn;

	IF g_tyNtParamCurr.bProjMag1ConvPrep THEN
		tylocalAGV.In.eAct := tyOpsMagConvUL1.eAGVMagAct;
	ELSIF g_tyNtParamCurr.bProjMagConvLane1Prep THEN
		//	tylocalAGV.In.eAct := tyOpsInMagConvAGVMagAct;
	ELSE
		tylocalAGV.In.eAct := eAct;
	END_IF

	IF EDGENEG(g_tyOps.bRun) THEN
		tylocalAGV.In.eAct	:= AGVMagActIdle;
	END_IF
END_ACTION
```

#### Act_Link.st
```iecst
(** 2018-12-08 **)
ACTION Act_Link:

	//Machine --> AGV ---> Communication On & Machine itself RUN Mode
	IF p_bLinkOpsRun = TRUE THEN

		tyDTMagToAGV.bCI1Auto := TRUE;
	ELSE
		tyDTMagToAGV.bCI1Auto	:= FALSE;
	END_IF

	tyDTMagToAGV.bCI1Occupied 			:= p_bBufferMagPresent OR p_bMagConvLftSen OR p_bMagConvRgtSen; // Magazine is present

	fbMagFullTm(IN:= p_bMagConvRgtSen = FALSE AND p_bBufferMagPresent = FALSE);
	IF p_bBufferMagPresent AND p_tyLinkBufferStat.bBffrFull THEN
		tyDTMagToAGV.bCI1MagazineFull		:=  TRUE;
	ELSIF fbMagFullTm.Q THEN
		tyDTMagToAGV.bCI1MagazineFull		:=  FALSE;
	END_IF

	IF p_bLinkAGVOnline THEN

		p_tyAGVToDTMag.bVEHAuto		:= p_tyLinkAGVtoDTMag.bVEHAuto;
		p_tyAGVToDTMag.bVEHInPos1	:= p_tyLinkAGVtoDTMag.bVEHInPos1 AND bAGVInPosSen;
		p_tyAGVToDTMag.bVEHInPos2 	:= p_tyLinkAGVtoDTMag.bVEHInPos2;
		p_tyAGVToDTMag.bVEHInPos3 	:= p_tyLinkAGVtoDTMag.bVEHInPos3;
		p_tyAGVToDTMag.bVEH1Occupied	:= p_tyLinkAGVtoDTMag.bVEH1Occupied;
		p_tyAGVToDTMag.bVEH2Occupied	:= p_tyLinkAGVtoDTMag.bVEH2Occupied;
		p_tyAGVToDTMag.bVEH3Occupied	:= p_tyLinkAGVtoDTMag.bVEH3Occupied;
		p_tyAGVToDTMag.bVEHRunning	:= p_tyLinkAGVtoDTMag.bVEHRunning;

	ELSE

		p_tyAGVToDTMag.bVEHAuto		:= FALSE;
		p_tyAGVToDTMag.bVEHInPos1	:= FALSE;
		p_tyAGVToDTMag.bVEHInPos2 	:= FALSE;
		p_tyAGVToDTMag.bVEHInPos3 	:= FALSE;
		p_tyAGVToDTMag.bVEH1Occupied:= FALSE;
		p_tyAGVToDTMag.bVEH2Occupied:= FALSE;
		p_tyAGVToDTMag.bVEH3Occupied:= FALSE;
		p_tyAGVToDTMag.bVEHRunning	:= FALSE;

	END_IF

	bAIVInPos := p_tyAGVToDTMag.bVEHInPos1;
	bAIVAuto := p_tyAGVToDTMag.bVEHAuto;
	bAIVOccupied := p_tyAGVToDTMag.bVEH1Occupied;
	bMagConvAuto := tyDTMagToAGV.bCI1Auto;
	bMagConvOccupied :=  tyDTMagToAGV.bCI1Occupied;

	tyDTMagToAGV.bCI1Running := bMagConvRun;
	tyDTMagToAGV.bCI1Rdy	:= bMagConvRdy;

	IF p_bNtParamAGVInPosSenPrep THEN
		fbInPosErrTimer(IN:= p_tyLinkAGVtoDTMag.bVEHInPos1 AND bAGVInPosSen = FALSE, PT:= T#10s);
		IF fbInPosErrTimer.Q THEN
			eStatus		:= Error;
			udiStatus	:= 10009;	//AIV Not In Position
		END_IF
	END_IF

	IF p_bNtParamAGVInPosSenPrep THEN
		bAGVInPosSen := p_bAGVInPosSen1 AND p_bAGVInPosSen2;
	ELSE
		bAGVInPosSen := TRUE;
	END_IF

END_ACTION
```

#### Act_LinkAction.st
```iecst
(** 2019-03-29 **)
ACTION Act_LinkAction:
	IF p_bLinkProjMag1ConvPrep THEN
		p_eAct ACCESS p_OpsMagConvUL1AGVMagAct;
	ELSIF p_bLinkProjMagConvLane1Prep THEN
	//	p_eAct ACCESS p_OpsInMagConvAGVMagAct;
	ELSE
		p_eAct ACCESS ADR(eAct);
	END_IF

	IF EDGENEG(p_bLinkOpsRun) THEN
		p_eAct	:= AGVMagActIdle;
	END_IF

END_ACTION
```

#### Act_OutputConfig.st
```iecst
ACTION Act_OutputConfig:

	g_tyAGV1 := tylocalAGV.Out; // Change the Global Naming According to the Physical Hardware Module

END_ACTION
```

#### Init.st
```iecst
(** 2019-01-20 **)
PROGRAM _INIT

	(* Always Change If Project Change *)

	sProgNm	:= 'AGVMag 1';

	//Physical Configuration

	//Pass Address To Global Address For External Use
	//Action, State & Status
	p_AGVMag1Stat			:= ADR(eStat);
	p_AGVMag1Status			:= ADR(eStatus);
	p_AGVMag1StatTxt		:= ADR(sStatTxt);

	//Alarm
	p_AGVMag1AlmData		:= ADR(tyAlmData);

	//Output
	p_AGVMag1RdyEnter		:= ADR(bRdyEnt);
	p_AGVMag1RdyExit		:= ADR(bRdyExit);
	p_AGVMag1McRunRdy		:= ADR(bMcRunRdy);
	p_AGVMag1DTMagToAGV		:= ADR(tyDTMagToAGV);

	(* Always Change If Project Change *)

END_PROGRAM
```

### Program Logical/AGVCom/AGV2 (IEC) - 1.00.0 - NtSMEMA v5.00.0

#### InputRef_Link.var
```iecst
(*2018-12-08*)
(**)
(*External Data*)
VAR
	p_bLinkAGVOnline : REFERENCE TO BOOL;
	p_bLinkOpsRun : REFERENCE TO BOOL;
END_VAR
(**)
VAR
	p_tyLinkBufferStat : REFERENCE TO tyBffrStat;
	p_tyLinkAGVtoDTMag : REFERENCE TO tyTagAGVToDTMag;
	p_bLinkProjMag2ConvPrep : REFERENCE TO BOOL;
	p_bLinkProjMagConvLane2Prep : REFERENCE TO BOOL;
END_VAR
```

#### Local.var
```iecst
(*2019-01-20*)
VAR
	tylocalAGV : tyAGV1;
END_VAR
(**)
(*Local Action, State & Status*)
VAR
	eAct : eAGVMagAction := AGVMagActIdle;
	eStat : eAGVMagAction := AGVMagActIdle;
	eStatus : eFBStatus := Idle;
	udiStatus : UDINT := 0;
	sStatTxt : STRING[100] := '';
	a_sStatText : ARRAY[0..50] OF STRING[100] := ['Idling','AIV Magazine Ready Enter And Communicating AIV','AIV Magazine Ready Exit And Communicating AIV',48('')];
END_VAR
(**)
(*Local Alarm*)
VAR
	tyAlmData : tyAlmDat;
	a_tyAlmText : ARRAY[10000..10099] OF tyAlmTxt := [(sAlmText:='Magazine Is Present Before Entering',sRcyText:='Remove Magazine To Continue Operation.'),(sAlmText:='AGV Not In Enter Position',sRcyText:='Adjust AGV Position And Restart Operation.'),(sAlmText:='Transfer In Time Out While Transporting',sRcyText:='Adjust Magazine Position Or Transporting Time Or Check Online Connection'),(sAlmText:='Magazine Is Not Present Before Exiting',sRcyText:='Magazine Has Taken Away, Restart Operation.'),(sAlmText:='AGV Not In Exit Position',sRcyText:='Adjust AGV Position And Restart Operation.'),(sAlmText:='Transfer Out Time Out While Transporting',sRcyText:='Adjust Magazine Position Or Transporting Time.'),(sAlmText:='AGV is not in Auto',sRcyText:='Make Sure AGV is in Auto'),(sAlmText:='Magazine is not Present in AGV while Entering',sRcyText:='Check AGV'),(sAlmText:='Magazine is Present in AGV while Exiting',sRcyText:='Check AGV'),(sAlmText:='AGV In Position Sensor is off while received the AGV in position signal',sRcyText:='Check AGV in position sensor'),(sAlmText:='SOT Error Signal Has Been Activated',sRcyText:='AIV Activated The Error Signal During Magazine Transportation'),89((0))];
END_VAR
(**)
(*Local Output*)
VAR
	bMcRunRdy : BOOL;
	bRdyEnt : BOOL;
	bRdyExit : BOOL;
	bMagEnt : BOOL;
	bMagExit : BOOL;
END_VAR
(*Local*)
VAR
	bRstErr : BOOL;
	udiRstErrOld : UDINT;
	bInitDone : BOOL;
	bInitialDone : BOOL;
	usiStep : USINT;
	bEndSen : BOOL;
	bAGVInPosSen : BOOL;
	fbMagFullTm : TON := (PT:=T#2s);
	fbInPosErrTimer : TON;
	fbTxInTimer : TON;
	fbTxOutTimer : TON;
	fbMagOutTrig : F_TRIG;
	eStatOld : eAGVMagAction := AGVMagActIdle;
	fbCheckErrorTim : TON := (PT:=T#1s);
	bMagConvRun : BOOL;
	bMagConvRdy : BOOL;
	bMagConvAuto : BOOL;
	bMagConvOccupied : BOOL;
	bAIVOccupied : BOOL;
	bAIVAuto : BOOL;
	bAIVInPos : BOOL;
	udiModuleNum : UDINT := 6161;
END_VAR
```

#### Act_Alarm.st
```iecst
(** 2019-03-25 **)
ACTION Act_Alarm:
	//Reset Error
	IF (tylocalAGV.Out.eStatus = Error) AND bRstErr THEN
		tylocalAGV.In.eAct	:= AGVMagActIdle;
		tylocalAGV.Out.eStat	:= AGVMagActIdle;
	END_IF

	//Error
	IF tylocalAGV.In.udiRstErr <> udiRstErrOld THEN
		bRstErr			:= TRUE;
		udiRstErrOld	:= tylocalAGV.In.udiRstErr;
	ELSE
		bRstErr			:= FALSE;
	END_IF

	IF EDGEPOS(tylocalAGV.Out.eStatus = Error) THEN

		tylocalAGV.Out.tyAlmData.sProgNm		:= tylocalAGV.In.sProgNm;
		tylocalAGV.Out.tyAlmData.udiCode		:= udiStatus;
		tylocalAGV.Out.tyAlmData.eSeverity		:= AlmSeverityError;
		tylocalAGV.Out.tyAlmData.udiRunTime	:= tylocalAGV.Out.tyAlmData.udiRunTime + 1;
		tylocalAGV.Out.tyAlmData.bAlm			:= TRUE;
		tylocalAGV.Out.tyAlmData.udiModuleNum  := udiModuleNum;
		g_sAGVProgNm		:= tylocalAGV.In.sProgNm;

		//Get Error Message
		IF tylocalAGV.Out.tyAlmData.udiCode < 10000 OR tylocalAGV.Out.tyAlmData.udiCode > 10099 THEN
			tylocalAGV.Out.tyAlmData.sAlmMsg	:= 'Unknown';
			tylocalAGV.Out.tyAlmData.sRcyMsg	:= 'Unknown';
		ELSE
			tylocalAGV.Out.tyAlmData.sAlmMsg	:= a_tyAlmText[tylocalAGV.Out.tyAlmData.udiCode].sAlmText;
			tylocalAGV.Out.tyAlmData.sRcyMsg	:= a_tyAlmText[tylocalAGV.Out.tyAlmData.udiCode].sRcyText;
		END_IF

		tylocalAGV.Out.sStatTxt	:= tylocalAGV.Out.tyAlmData.sAlmMsg;

	ELSIF bRstErr AND (tylocalAGV.Out.tyAlmData.udiCode <> 0) THEN

		tylocalAGV.Out.tyAlmData.udiCode	:= 0;
		tylocalAGV.Out.tyAlmData.eSeverity	:= AlmSeverityNA;
		tylocalAGV.Out.tyAlmData.sAlmMsg	:= '';
		tylocalAGV.Out.tyAlmData.sRcyMsg	:= '';
		tylocalAGV.Out.tyAlmData.bAlm			:= FALSE;
		tylocalAGV.Out.sStatTxt	:= a_sStatText[tylocalAGV.Out.eStat];

	END_IF

END_ACTION
```

#### Act_Background.st
```iecst
(** 2019-01-20 **)
ACTION Act_Background:

END_ACTION
```

#### Act_InitGlobal.st
```iecst
(** 2018-12-08 **)
ACTION Act_InitGlobal:

	(* Always Change If Project Change *)

	//Pass Data To Link
	p_bLinkOpsRun ACCESS p_OpsRun;

	p_tyLinkBufferStat ACCESS p_Buffer2BffrStat;
	p_bLinkAGVOnline ACCESS p_AGVOnline;
	p_tyLinkAGVtoDTMag ACCESS p_AGVTagAGVToDTMag;
	p_bLinkProjMag2ConvPrep ACCESS p_NtParamProjMag2ConvPrep;
	p_bLinkProjMagConvLane2Prep ACCESS p_NtParamProjMagConvLane2Prep;

	//Pass Data To Internal Use
//	p_eAct ACCESS p_OpsMagConvUL2AGVMagAct;
	p_udiRstErr	ACCESS p_RstErrReset;
	p_bPrep ACCESS p_NtParamProjAGVPrep;
	p_sProgNm ACCESS p_NtParamAGVMag2ProgNm;
	p_diTxInTimeOut ACCESS p_McParamMag2ConvRunTmOut;
	p_diTxOutTimeOut ACCESS p_McParamMag2ConvRunTmOut;
	p_eDirection ACCESS p_NtParamProjMagConvDir;
	p_bBufferMagPresent ACCESS p_DIMagPresentSen2;
	p_bMagConvLftSen ACCESS p_DIMagPresentSen2;
	p_bMagConvRgtSen ACCESS p_DIMagConvEntSen2;
	p_bMagConvMtrIn ACCESS p_MagConv2Clp2MtrSigOnOrLToR;
	p_bMagConvMtrOut ACCESS p_MagConv2Clp2MtrDirOrRToL;
	p_bNtSettingsLoadDone ACCESS p_StartupNtSettingsLoadDone;
	p_bAGVInPosSen1	ACCESS p_DIMag2AIVInPosSen1;
	p_bAGVInPosSen2	ACCESS p_DIMag2AIVInPosSen2;
	p_bNtParamAGVInPosSenPrep ACCESS p_NtParamProjAIVInPosSenPrep;
	p_bSOTRcvOk ACCESS p_DISOT2Receive;
	p_bSOTErr ACCESS p_DISOT2Error;
	p_bSOTRdy ACCESS p_DISOT2Ready;
	p_bSOTAvailable ACCESS p_DISOT2Available;
	p_bEn ACCESS p_McParamAGVComEn;
	(* Always Change If Project Change *)

END_ACTION
```

#### Act_Initial.st
```iecst
(** 2019-01-12 **)
ACTION Act_Initial:

	//Initial
	sStatTxt	:= a_sStatText[eStat];

	fbTxInTimer(IN := FALSE);
	fbTxOutTimer(IN := FALSE);
	fbMagOutTrig(CLK := FALSE);

	tylocalAGV.Out.bMcRunRdy			:= FALSE;
	tylocalAGV.Out.bRdyEnt			 	:= FALSE;
	tylocalAGV.Out.bRdyExit				:= FALSE;
	tylocalAGV.Out.bMagConvRun	    	:= FALSE;

END_ACTION
```

#### Act_InputConfig.st
```iecst
ACTION Act_InputConfig:

	(* Always Change If Project Change *)

	//Pass Data To Link
	tylocalAGV.In.bLinkOpsRun := g_tyOps.bRun;

	tylocalAGV.In.tyLinkBufferStat := g_tyBuffer2.tyBufferStat;
	tylocalAGV.In.bLinkAGVOnline := g_tyAGV.bInternalAGVOnline;
	tylocalAGV.In.tyLinkAGVtoDTMag := g_tyAGV.tyAGVToDTMag;

	//Pass Data To Internal Use
//	tylocalAGV.In.eAct := g_tyOpsMagConvUL2AGVMagAct;
	tylocalAGV.In.udiRstErr	:= g_tyRstErrOut.udiRstErr;
	tylocalAGV.In.bPrep := g_tyNtParamCurr.bProjAGVPrep;
	tylocalAGV.In.sProgNm := g_tyNtParamCurr.sAGVMag2ProgNm;

	tylocalAGV.In.diTxInTimeOut := g_tyMcParam.tMag2ConvRunTmOut;
	tylocalAGV.In.diTxOutTimeOut := g_tyMcParam.tMag2ConvRunTmOut;

	tylocalAGV.In.eDirection := g_tyNtParamCurr.bProjMagConvDir;
	tylocalAGV.In.bBufferMagPresent := g_tyDInput.bMagPresentSen2;
	tylocalAGV.In.bMagConvLftSen := g_tyDInput.bMagPresentSen2;
	tylocalAGV.In.bMagConvRgtSen := g_tyDInput.bMagConvEntSen2;
	tylocalAGV.In.bMagConvMtrIn := g_tyMagConv2Clp2.bMtrSigOnOrLToR;
	tylocalAGV.In.bMagConvMtrOut := g_tyMagConv2Clp2.bMtrDirOrRToL;

	tylocalAGV.In.bAGVInPosSen1	:= g_tyDInput.bMag2AIVInPosSen1;
	tylocalAGV.In.bAGVInPosSen2	:= g_tyDInput.bMag2AIVInPosSen2;

	tylocalAGV.In.bNtParamAGVInPosSenPrep := g_tyNtParamCurr.bProjAIVInPosSenPrep;

	tylocalAGV.In.bSOTRcvOk := g_tyDInput.bSOT2Receive;
	tylocalAGV.In.bSOTErr := g_tyDInput.bSOT2AIVError;
	tylocalAGV.In.bSOTRdy := g_tyDInput.bSOT2AIVReady;
	tylocalAGV.In.bSOTAvailable := g_tyDInput.bSOT2AIVAvailable;
	tylocalAGV.In.bEn := g_tyMcParam.AGVComEn;

	IF g_tyNtParamCurr.bProjMag2ConvPrep THEN
		tylocalAGV.In.eAct := tyOpsMagConvUL2.eAGVMagAct;
	ELSIF g_tyNtParamCurr.bProjMagConvLane2Prep THEN
		//	tylocalAGV.In.eAct := tyOpsInMagConvAGVMagAct;
	ELSE
		tylocalAGV.In.eAct := eAct;
	END_IF

	IF EDGENEG(g_tyOps.bRun) THEN
		tylocalAGV.In.eAct	:= AGVMagActIdle;
	END_IF
END_ACTION
```

#### Act_Link.st
```iecst
(** 2018-12-08 **)
ACTION Act_Link:

	//Machine --> AGV ---> Communication On & Machine itself RUN Mode
	IF g_tyOps.bRun = TRUE THEN

		tylocalAGV.Out.tyDTMagToAGV.bCI1Auto := TRUE;
	ELSE
		tylocalAGV.Out.tyDTMagToAGV.bCI1Auto	:= FALSE;
	END_IF

	tylocalAGV.Out.tyDTMagToAGV.bCI1Occupied 			:= tylocalAGV.In.bBufferMagPresent OR tylocalAGV.In.bMagConvLftSen OR tylocalAGV.In.bMagConvRgtSen; // Magazine is present

	fbMagFullTm(IN:= tylocalAGV.In.bMagConvRgtSen = FALSE AND tylocalAGV.In.bBufferMagPresent = FALSE);
	IF tylocalAGV.In.bBufferMagPresent AND tylocalAGV.In.tyLinkBufferStat.bBffrFull THEN
		tylocalAGV.Out.tyDTMagToAGV.bCI1MagazineFull		:=  TRUE;
	ELSIF fbMagFullTm.Q THEN
		tylocalAGV.Out.tyDTMagToAGV.bCI1MagazineFull		:=  FALSE;
	END_IF

	IF tylocalAGV.In.bLinkAGVOnline THEN

		tylocalAGV.In.tyAGVToDTMag.bVEHAuto		:= tylocalAGV.In.tyLinkAGVtoDTMag.bVEHAuto;
		tylocalAGV.In.tyAGVToDTMag.bVEHInPos1	:= tylocalAGV.In.tyLinkAGVtoDTMag.bVEHInPos1 AND bAGVInPosSen;
		tylocalAGV.In.tyAGVToDTMag.bVEHInPos2 	:= tylocalAGV.In.tyLinkAGVtoDTMag.bVEHInPos2;
		tylocalAGV.In.tyAGVToDTMag.bVEHInPos3 	:= tylocalAGV.In.tyLinkAGVtoDTMag.bVEHInPos3;
		tylocalAGV.In.tyAGVToDTMag.bVEH1Occupied	:= tylocalAGV.In.tyLinkAGVtoDTMag.bVEH1Occupied;
		tylocalAGV.In.tyAGVToDTMag.bVEH2Occupied	:= tylocalAGV.In.tyLinkAGVtoDTMag.bVEH2Occupied;
		tylocalAGV.In.tyAGVToDTMag.bVEH3Occupied	:= tylocalAGV.In.tyLinkAGVtoDTMag.bVEH3Occupied;
		tylocalAGV.In.tyAGVToDTMag.bVEHRunning	:= tylocalAGV.In.tyLinkAGVtoDTMag.bVEHRunning;

	ELSE

		tylocalAGV.In.tyAGVToDTMag.bVEHAuto		:= FALSE;
		tylocalAGV.In.tyAGVToDTMag.bVEHInPos1	:= FALSE;
		tylocalAGV.In.tyAGVToDTMag.bVEHInPos2 	:= FALSE;
		tylocalAGV.In.tyAGVToDTMag.bVEHInPos3 	:= FALSE;
		tylocalAGV.In.tyAGVToDTMag.bVEH1Occupied:= FALSE;
		tylocalAGV.In.tyAGVToDTMag.bVEH2Occupied:= FALSE;
		tylocalAGV.In.tyAGVToDTMag.bVEH3Occupied:= FALSE;
		tylocalAGV.In.tyAGVToDTMag.bVEHRunning	:= FALSE;

	END_IF

	bAIVInPos := tylocalAGV.In.tyAGVToDTMag.bVEHInPos1;
	bAIVAuto := tylocalAGV.In.tyAGVToDTMag.bVEHAuto;
	bAIVOccupied := tylocalAGV.In.tyAGVToDTMag.bVEH1Occupied;
	bMagConvAuto := tylocalAGV.Out.tyDTMagToAGV.bCI1Auto;
	bMagConvOccupied :=  tylocalAGV.Out.tyDTMagToAGV.bCI1Occupied;

	tylocalAGV.Out.tyDTMagToAGV.bCI1Running := bMagConvRun;
	tylocalAGV.Out.tyDTMagToAGV.bCI1Rdy	:= bMagConvRdy;

	IF tylocalAGV.In.bNtParamAGVInPosSenPrep THEN
		fbInPosErrTimer(IN:= tylocalAGV.In.tyLinkAGVtoDTMag.bVEHInPos1 AND bAGVInPosSen = FALSE, PT:= T#10s);
		IF fbInPosErrTimer.Q THEN
			tylocalAGV.Out.eStatus		:= Error;
			udiStatus	:= 10009;	//AIV Not In Position
		END_IF
	END_IF

	IF tylocalAGV.In.bNtParamAGVInPosSenPrep THEN
		bAGVInPosSen := tylocalAGV.In.bAGVInPosSen1 AND tylocalAGV.In.bAGVInPosSen2;
	ELSE
		bAGVInPosSen := TRUE;
	END_IF

END_ACTION
```

#### Act_LinkAction.st
```iecst
(** 2019-03-29 **)
ACTION Act_LinkAction:
	IF p_bLinkProjMag2ConvPrep THEN
		p_eAct ACCESS p_OpsMagConvUL2AGVMagAct;
	ELSIF p_bLinkProjMagConvLane2Prep THEN
	//	p_eAct ACCESS p_OpsInMagConv2AGVMagAct;
	ELSE
		p_eAct ACCESS ADR(eAct);
	END_IF

	IF EDGENEG(p_bLinkOpsRun) THEN
		p_eAct	:= AGVMagActIdle;
	END_IF

END_ACTION
```
